LIN {X 0,Y 385.794,Z 704.121,A -85,B 0,C 180,E1 11186.142,E2 11186.142} C_VEL
LIN {X 0,Y 379.875,Z 692.265,A -85,B 0,C 180,E1 11183.296,E2 11183.296} C_VEL
LIN {X 0,Y 374.459,Z 681.957,A -85,B 0,C 180,E1 11180.23,E2 11180.23} C_VEL
LIN {X 0,Y 370.594,Z 674.701,A -85,B 0,C 180,E1 11177.589,E2 11177.589} C_VEL
LIN {X 0,Y 366.819,Z 667.673,A -85,B 0,C 180,E1 11174.362,E2 11174.362} C_VEL
LIN {X 0,Y 365.103,Z 664.56,A -85,B 0,C 180,E1 11172.495,E2 11172.495} C_VEL
LIN {X 0,Y 363.524,Z 661.381,A -85,B 0,C 180,E1 11170.299,E2 11170.299} C_VEL
LIN {X 0,Y 361.927,Z 657.573,A -85,B 0,C 180,E1 11166.663,E2 11166.663} C_VEL
LIN {X 0,Y 361.691,Z 655.978,A -85,B 0,C 180,E1 11161.584,E2 11161.584} C_VEL
LIN {X 0,Y 363.057,Z 656.603,A -85,B 0,C 180,E1 11157.948,E2 11157.948} C_VEL
LIN {X 0,Y 366.472,Z 659.778,A -85,B 0,C 180,E1 11153.498,E2 11153.498} C_VEL
LIN {X 0,Y 370.493,Z 664.801,A -85,B 0,C 180,E1 11149.975,E2 11149.975} C_VEL
LIN {X 0,Y 374.313,Z 669.836,A -85,B 0,C 180,E1 11147.347,E2 11147.347} C_VEL
LIN {X 0,Y 379.523,Z 676.993,A -85,B 0,C 180,E1 11144.372,E2 11144.372} C_VEL
LIN {X 0,Y 385.577,Z 686.162,A -85,B 0,C 180,E1 11141.439,E2 11141.439} C_VEL
LIN {X 0,Y 391.936,Z 696.414,A -85,B 0,C 180,E1 11138.761,E2 11138.761} C_VEL
LIN {X 0,Y 396.859,Z 705.085,A -85,B 0,C 180,E1 11136.889,E2 11136.889} C_VEL
LIN {X 0,Y 378.142,Z 929.621,A -85,B 0,C 180,E1 11132.962,E2 11132.962} C_VEL
LIN {X 0,Y 374.66,Z 954.802,A -85,B 0,C 180,E1 11132.348,E2 11132.348} C_VEL
LIN {X 0,Y 370.716,Z 975.799,A -85,B 0,C 180,E1 11131.66,E2 11131.66} C_VEL
LIN {X 0,Y 365.231,Z 998.846,A -85,B 0,C 180,E1 11130.683,E2 11130.683} C_VEL
LIN {X 0,Y 359.243,Z 1019.879,A -85,B 0,C 180,E1 11129.564,E2 11129.564} C_VEL
LIN {X 0,Y 351.998,Z 1041.518,A -85,B 0,C 180,E1 11128.137,E2 11128.137} C_VEL
LIN {X 0,Y 344.181,Z 1062.128,A -85,B 0,C 180,E1 11126.485,E2 11126.485} C_VEL
LIN {X 0,Y 335.714,Z 1081.84,A -85,B 0,C 180,E1 11124.544,E2 11124.544} C_VEL
LIN {X 0,Y 327.05,Z 1100.424,A -85,B 0,C 180,E1 11122.355,E2 11122.355} C_VEL
LIN {X 0,Y 318.011,Z 1118.05,A -85,B 0,C 180,E1 11119.819,E2 11119.819} C_VEL
LIN {X 0,Y 308.974,Z 1134.8,A -85,B 0,C 180,E1 11116.934,E2 11116.934} C_VEL
LIN {X 0,Y 300.211,Z 1150.077,A -85,B 0,C 180,E1 11113.718,E2 11113.718} C_VEL
LIN {X 0,Y 291.457,Z 1165.019,A -85,B 0,C 180,E1 11109.905,E2 11109.905} C_VEL
LIN {X 0,Y 284.438,Z 1176.9,A -85,B 0,C 180,E1 11106.196,E2 11106.196} C_VEL
LIN {X 0,Y 277.366,Z 1189.144,A -85,B 0,C 180,E1 11101.514,E2 11101.514} C_VEL
LIN {X 0,Y 272.523,Z 1198.075,A -85,B 0,C 180,E1 11097.297,E2 11097.297} C_VEL
LIN {X 0,Y 268.421,Z 1206.484,A -85,B 0,C 180,E1 11092.33,E2 11092.33} C_VEL
LIN {X 0,Y 266.058,Z 1212.321,A -85,B 0,C 180,E1 11087.948,E2 11087.948} C_VEL
LIN {X 0,Y 264.493,Z 1217.601,A -85,B 0,C 180,E1 11082.665,E2 11082.665} C_VEL
LIN {X 0,Y 264.031,Z 1220.449,A -85,B 0,C 180,E1 11078.493,E2 11078.493} C_VEL
LIN {X 0,Y 263.961,Z 1222.135,A -85,B 0,C 180,E1 11074.562,E2 11074.562} C_VEL
LIN {X 0,Y 264,Z 1222.893,A -85,B 0,C 180,E1 11070,E2 11070} C_VEL
LIN {X 0,Y 263.966,Z 1222.194,A -85,B 0,C 180,E1 11065.655,E2 11065.655} C_VEL
LIN {X 0,Y 264.013,Z 1220.547,A -85,B 0,C 180,E1 11061.726,E2 11061.726} C_VEL
LIN {X 0,Y 264.454,Z 1217.74,A -85,B 0,C 180,E1 11057.555,E2 11057.555} C_VEL
LIN {X 0,Y 265.965,Z 1212.541,A -85,B 0,C 180,E1 11052.271,E2 11052.271} C_VEL
LIN {X 0,Y 268.274,Z 1206.745,A -85,B 0,C 180,E1 11047.888,E2 11047.888} C_VEL
LIN {X 0,Y 272.305,Z 1198.419,A -85,B 0,C 180,E1 11042.915,E2 11042.915} C_VEL
LIN {X 0,Y 277.088,Z 1189.533,A -85,B 0,C 180,E1 11038.694,E2 11038.694} C_VEL
LIN {X 0,Y 283.752,Z 1177.976,A -85,B 0,C 180,E1 11034.202,E2 11034.202} C_VEL
LIN {X 0,Y 290.655,Z 1166.202,A -85,B 0,C 180,E1 11030.476,E2 11030.476} C_VEL
LIN {X 0,Y 299.51,Z 1151.115,A -85,B 0,C 180,E1 11026.553,E2 11026.553} C_VEL
LIN {X 0,Y 307.569,Z 1137.016,A -85,B 0,C 180,E1 11023.536,E2 11023.536} C_VEL
LIN {X 0,Y 317.175,Z 1119.387,A -85,B 0,C 180,E1 11020.421,E2 11020.421} C_VEL
LIN {X 0,Y 325.578,Z 1103.038,A -85,B 0,C 180,E1 11018.027,E2 11018.027} C_VEL
LIN {X 0,Y 334.775,Z 1083.58,A -85,B 0,C 180,E1 11015.672,E2 11015.672} C_VEL
LIN {X 0,Y 342.885,Z 1064.882,A -85,B 0,C 180,E1 11013.792,E2 11013.792} C_VEL
LIN {X 0,Y 350.98,Z 1043.855,A -85,B 0,C 180,E1 11012.059,E2 11012.059} C_VEL
LIN {X 0,Y 358.352,Z 1022.299,A -85,B 0,C 180,E1 11010.598,E2 11010.598} C_VEL
LIN {X 0,Y 364.543,Z 1000.723,A -85,B 0,C 180,E1 11009.429,E2 11009.429} C_VEL
LIN {X 0,Y 370.058,Z 978.122,A -85,B 0,C 180,E1 11008.442,E2 11008.442} C_VEL
LIN {X 0,Y 374.312,Z 955.693,A -85,B 0,C 180,E1 11007.695,E2 11007.695} C_VEL
LIN {X 0,Y 377.785,Z 931.228,A -85,B 0,C 180,E1 11007.087,E2 11007.087} C_VEL
LIN {X 0,Y 387.415,Z 815.943,A -85,B 0,C 180,E1 11005.031,E2 11005.031} C_VEL
LIN {X 0,Y 396.675,Z 704.702,A -85,B 0,C 180,E1 11003.116,E2 11003.116} C_VEL
LIN {X 0,Y 389.19,Z 691.96,A -85,B 0,C 180,E1 11000.216,E2 11000.216} C_VEL
LIN {X 0,Y 382.087,Z 680.857,A -85,B 0,C 180,E1 10997.043,E2 10997.043} C_VEL
LIN {X 0,Y 376.158,Z 672.371,A -85,B 0,C 180,E1 10993.92,E2 10993.92} C_VEL
LIN {X 0,Y 372.332,Z 667.309,A -85,B 0,C 180,E1 10991.541,E2 10991.541} C_VEL
LIN {X 0,Y 369.337,Z 663.423,A -85,B 0,C 180,E1 10989.348,E2 10989.348} C_VEL
LIN {X 0,Y 365.813,Z 659.038,A -85,B 0,C 180,E1 10986.119,E2 10986.119} C_VEL
LIN {X 0,Y 362.366,Z 655.946,A -85,B 0,C 180,E1 10981.265,E2 10981.265} C_VEL
LIN {X 0,Y 361.292,Z 655.603,A -85,B 0,C 180,E1 10977.938,E2 10977.938} C_VEL
LIN {X 0,Y 361.77,Z 657.568,A -85,B 0,C 180,E1 10972.696,E2 10972.696} C_VEL
LIN {X 0,Y 363.871,Z 662.416,A -85,B 0,C 180,E1 10968.589,E2 10968.589} C_VEL
LIN {X 0,Y 366.53,Z 667.359,A -85,B 0,C 180,E1 10965.545,E2 10965.545} C_VEL
LIN {X 0,Y 370.214,Z 674.259,A -85,B 0,C 180,E1 10962.392,E2 10962.392} C_VEL
LIN {X 0,Y 373.963,Z 681.257,A -85,B 0,C 180,E1 10959.823,E2 10959.823} C_VEL
LIN {X 0,Y 377.627,Z 688.285,A -85,B 0,C 180,E1 10957.668,E2 10957.668} C_VEL
LIN {X 0,Y 382.471,Z 697.632,A -85,B 0,C 180,E1 10955.191,E2 10955.191} C_VEL
LIN {X 0,Y 388.587,Z 710.276,A -85,B 0,C 180,E1 10952.45,E2 10952.45} C_VEL
LIN {X 0,Y 391.861,Z 717.757,A -85,B 0,C 180,E1 10951.102,E2 10951.102} C_VEL
LIN {X 0,Y 392.576,Z 738.553,A -85,B 0,C 180,E1 10950.077,E2 10950.077} C_VEL
LIN {X 0,Y 377.124,Z 944.509,A -85,B 0,C 180,E1 10946.703,E2 10946.703} C_VEL
LIN {X 0,Y 373.9,Z 967.663,A -85,B 0,C 180,E1 10946.174,E2 10946.174} C_VEL
LIN {X 0,Y 369.642,Z 989.416,A -85,B 0,C 180,E1 10945.52,E2 10945.52} C_VEL
LIN {X 0,Y 364.143,Z 1011.031,A -85,B 0,C 180,E1 10944.636,E2 10944.636} C_VEL
LIN {X 0,Y 357.235,Z 1033.546,A -85,B 0,C 180,E1 10943.444,E2 10943.444} C_VEL
LIN {X 0,Y 350.094,Z 1053.415,A -85,B 0,C 180,E1 10942.117,E2 10942.117} C_VEL
LIN {X 0,Y 342.071,Z 1072.713,A -85,B 0,C 180,E1 10940.503,E2 10940.503} C_VEL
LIN {X 0,Y 333.358,Z 1091.539,A -85,B 0,C 180,E1 10938.576,E2 10938.576} C_VEL
LIN {X 0,Y 324.769,Z 1108.217,A -85,B 0,C 180,E1 10936.471,E2 10936.471} C_VEL
LIN {X 0,Y 315.047,Z 1125.58,A -85,B 0,C 180,E1 10933.778,E2 10933.778} C_VEL
LIN {X 0,Y 306.311,Z 1140.176,A -85,B 0,C 180,E1 10931.003,E2 10931.003} C_VEL
LIN {X 0,Y 297.865,Z 1153.372,A -85,B 0,C 180,E1 10927.9,E2 10927.9} C_VEL
LIN {X 0,Y 289.948,Z 1165.474,A -85,B 0,C 180,E1 10924.44,E2 10924.44} C_VEL
LIN {X 0,Y 282.737,Z 1176.152,A -85,B 0,C 180,E1 10920.613,E2 10920.613} C_VEL
LIN {X 0,Y 275.962,Z 1186.354,A -85,B 0,C 180,E1 10916.002,E2 10916.002} C_VEL
LIN {X 0,Y 271.018,Z 1194.256,A -85,B 0,C 180,E1 10911.422,E2 10911.422} C_VEL
LIN {X 0,Y 267.53,Z 1200.274,A -85,B 0,C 180,E1 10906.725,E2 10906.725} C_VEL
LIN {X 0,Y 265.265,Z 1205.087,A -85,B 0,C 180,E1 10901.524,E2 10901.524} C_VEL
LIN {X 0,Y 264.328,Z 1207.797,A -85,B 0,C 180,E1 10896.952,E2 10896.952} C_VEL
LIN {X 0,Y 264.041,Z 1209.184,A -85,B 0,C 180,E1 10892.17,E2 10892.17} C_VEL
LIN {X 0,Y 264.03,Z 1209.24,A -85,B 0,C 180,E1 10888.264,E2 10888.264} C_VEL
LIN {X 0,Y 264.252,Z 1208.179,A -85,B 0,C 180,E1 10883.7,E2 10883.7} C_VEL
LIN {X 0,Y 265.114,Z 1205.486,A -85,B 0,C 180,E1 10878.911,E2 10878.911} C_VEL
LIN {X 0,Y 267.122,Z 1201.154,A -85,B 0,C 180,E1 10873.92,E2 10873.92} C_VEL
LIN {X 0,Y 270.39,Z 1195.311,A -85,B 0,C 180,E1 10869.207,E2 10869.207} C_VEL
LIN {X 0,Y 275.363,Z 1187.374,A -85,B 0,C 180,E1 10864.399,E2 10864.399} C_VEL
LIN {X 0,Y 281.45,Z 1178.27,A -85,B 0,C 180,E1 10860.094,E2 10860.094} C_VEL
LIN {X 0,Y 288.655,Z 1167.471,A -85,B 0,C 180,E1 10856.105,E2 10856.105} C_VEL
LIN {X 0,Y 297.278,Z 1154.456,A -85,B 0,C 180,E1 10852.256,E2 10852.256} C_VEL
LIN {X 0,Y 306.152,Z 1140.649,A -85,B 0,C 180,E1 10848.971,E2 10848.971} C_VEL
LIN {X 0,Y 314.878,Z 1126.108,A -85,B 0,C 180,E1 10846.193,E2 10846.193} C_VEL
LIN {X 0,Y 324.307,Z 1109.391,A -85,B 0,C 180,E1 10843.571,E2 10843.571} C_VEL
LIN {X 0,Y 332.882,Z 1092.803,A -85,B 0,C 180,E1 10841.456,E2 10841.456} C_VEL
LIN {X 0,Y 341.882,Z 1073.546,A -85,B 0,C 180,E1 10839.459,E2 10839.459} C_VEL
LIN {X 0,Y 349.998,Z 1054.168,A -85,B 0,C 180,E1 10837.825,E2 10837.825} C_VEL
LIN {X 0,Y 357.378,Z 1033.67,A -85,B 0,C 180,E1 10836.452,E2 10836.452} C_VEL
LIN {X 0,Y 364.292,Z 1011.192,A -85,B 0,C 180,E1 10835.261,E2 10835.261} C_VEL
LIN {X 0,Y 369.611,Z 990.338,A -85,B 0,C 180,E1 10834.404,E2 10834.404} C_VEL
LIN {X 0,Y 374.035,Z 968.047,A -85,B 0,C 180,E1 10833.728,E2 10833.728} C_VEL
LIN {X 0,Y 377.274,Z 945.089,A -85,B 0,C 180,E1 10833.2,E2 10833.2} C_VEL
LIN {X 0,Y 385.345,Z 837.315,A -85,B 0,C 180,E1 10831.408,E2 10831.408} C_VEL
LIN {X 0,Y 392.815,Z 736.753,A -85,B 0,C 180,E1 10829.76,E2 10829.76} C_VEL
LIN {X 0,Y 392.625,Z 732.027,A -85,B 0,C 180,E1 10829.521,E2 10829.521} C_VEL
LIN {X 0,Y 392.068,Z 728.255,A -85,B 0,C 180,E1 10829.205,E2 10829.205} C_VEL
LIN {X 0,Y 390.556,Z 724.358,A -85,B 0,C 180,E1 10828.585,E2 10828.585} C_VEL
LIN {X 0,Y 386.327,Z 717.157,A -85,B 0,C 180,E1 10826.909,E2 10826.909} C_VEL
LIN {X 0,Y 380.447,Z 704.585,A -85,B 0,C 180,E1 10824.164,E2 10824.164} C_VEL
LIN {X 0,Y 375.315,Z 694.392,A -85,B 0,C 180,E1 10821.407,E2 10821.407} C_VEL
LIN {X 0,Y 371.624,Z 687.152,A -85,B 0,C 180,E1 10819.081,E2 10819.081} C_VEL
LIN {X 0,Y 368.331,Z 680.76,A -85,B 0,C 180,E1 10816.634,E2 10816.634} C_VEL
LIN {X 0,Y 364.751,Z 673.725,A -85,B 0,C 180,E1 10813.232,E2 10813.232} C_VEL
LIN {X 0,Y 362.352,Z 669.116,A -85,B 0,C 180,E1 10810.012,E2 10810.012} C_VEL
LIN {X 0,Y 360.908,Z 665.464,A -85,B 0,C 180,E1 10806.522,E2 10806.522} C_VEL
LIN {X 0,Y 360.716,Z 663.92,A -85,B 0,C 180,E1 10801.588,E2 10801.588} C_VEL
LIN {X 0,Y 362.079,Z 664.569,A -85,B 0,C 180,E1 10797.943,E2 10797.943} C_VEL
LIN {X 0,Y 365.256,Z 667.574,A -85,B 0,C 180,E1 10793.713,E2 10793.713} C_VEL
LIN {X 0,Y 369.182,Z 672.629,A -85,B 0,C 180,E1 10790.176,E2 10790.176} C_VEL
LIN {X 0,Y 372.704,Z 677.357,A -85,B 0,C 180,E1 10787.685,E2 10787.685} C_VEL
LIN {X 0,Y 377.735,Z 684.444,A -85,B 0,C 180,E1 10784.729,E2 10784.729} C_VEL
LIN {X 0,Y 383.502,Z 693.396,A -85,B 0,C 180,E1 10781.846,E2 10781.846} C_VEL
LIN {X 0,Y 389.565,Z 703.408,A -85,B 0,C 180,E1 10779.216,E2 10779.216} C_VEL
LIN {X 0,Y 392.961,Z 709.665,A -85,B 0,C 180,E1 10777.857,E2 10777.857} C_VEL
LIN {X 0,Y 374.215,Z 929.569,A -85,B 0,C 180,E1 10774.027,E2 10774.027} C_VEL
LIN {X 0,Y 370.645,Z 954.977,A -85,B 0,C 180,E1 10773.413,E2 10773.413} C_VEL
LIN {X 0,Y 366.64,Z 975.871,A -85,B 0,C 180,E1 10772.734,E2 10772.734} C_VEL
LIN {X 0,Y 360.947,Z 999.256,A -85,B 0,C 180,E1 10771.75,E2 10771.75} C_VEL
LIN {X 0,Y 355.065,Z 1019.451,A -85,B 0,C 180,E1 10770.685,E2 10770.685} C_VEL
LIN {X 0,Y 347.402,Z 1041.849,A -85,B 0,C 180,E1 10769.217,E2 10769.217} C_VEL
LIN {X 0,Y 339.431,Z 1062.322,A -85,B 0,C 180,E1 10767.579,E2 10767.579} C_VEL
LIN {X 0,Y 330.689,Z 1082.093,A -85,B 0,C 180,E1 10765.632,E2 10765.632} C_VEL
LIN {X 0,Y 321.475,Z 1101.221,A -85,B 0,C 180,E1 10763.363,E2 10763.363} C_VEL
LIN {X 0,Y 312.175,Z 1118.751,A -85,B 0,C 180,E1 10760.813,E2 10760.813} C_VEL
LIN {X 0,Y 302.457,Z 1136.035,A -85,B 0,C 180,E1 10757.774,E2 10757.774} C_VEL
LIN {X 0,Y 293.558,Z 1150.996,A -85,B 0,C 180,E1 10754.558,E2 10754.558} C_VEL
LIN {X 0,Y 284.306,Z 1166.072,A -85,B 0,C 180,E1 10750.588,E2 10750.588} C_VEL
LIN {X 0,Y 276.716,Z 1178.428,A -85,B 0,C 180,E1 10746.598,E2 10746.598} C_VEL
LIN {X 0,Y 270.039,Z 1189.39,A -85,B 0,C 180,E1 10742.221,E2 10742.221} C_VEL
LIN {X 0,Y 264.749,Z 1198.691,A -85,B 0,C 180,E1 10737.679,E2 10737.679} C_VEL
LIN {X 0,Y 260.66,Z 1206.584,A -85,B 0,C 180,E1 10732.794,E2 10732.794} C_VEL
LIN {X 0,Y 258.073,Z 1212.639,A -85,B 0,C 180,E1 10728.056,E2 10728.056} C_VEL
LIN {X 0,Y 256.518,Z 1217.562,A -85,B 0,C 180,E1 10722.837,E2 10722.837} C_VEL
LIN {X 0,Y 256.034,Z 1220.362,A -85,B 0,C 180,E1 10718.534,E2 10718.534} C_VEL
LIN {X 0,Y 255.964,Z 1222.002,A -85,B 0,C 180,E1 10714.481,E2 10714.481} C_VEL
LIN {X 0,Y 256.002,Z 1222.689,A -85,B 0,C 180,E1 10710,E2 10710} C_VEL
LIN {X 0,Y 255.964,Z 1221.989,A -85,B 0,C 180,E1 10705.519,E2 10705.519} C_VEL
LIN {X 0,Y 256.034,Z 1220.34,A -85,B 0,C 180,E1 10701.466,E2 10701.466} C_VEL
LIN {X 0,Y 256.547,Z 1217.411,A -85,B 0,C 180,E1 10697.002,E2 10697.002} C_VEL
LIN {X 0,Y 258.235,Z 1212.14,A -85,B 0,C 180,E1 10691.559,E2 10691.559} C_VEL
LIN {X 0,Y 260.857,Z 1206.118,A -85,B 0,C 180,E1 10686.919,E2 10686.919} C_VEL
LIN {X 0,Y 265.42,Z 1197.347,A -85,B 0,C 180,E1 10681.663,E2 10681.663} C_VEL
LIN {X 0,Y 270.607,Z 1188.348,A -85,B 0,C 180,E1 10677.354,E2 10677.354} C_VEL
LIN {X 0,Y 277.762,Z 1176.54,A -85,B 0,C 180,E1 10672.789,E2 10672.789} C_VEL
LIN {X 0,Y 285.492,Z 1164.055,A -85,B 0,C 180,E1 10668.852,E2 10668.852} C_VEL
LIN {X 0,Y 294.012,Z 1150.038,A -85,B 0,C 180,E1 10665.255,E2 10665.255} C_VEL
LIN {X 0,Y 302.957,Z 1134.986,A -85,B 0,C 180,E1 10662.049,E2 10662.049} C_VEL
LIN {X 0,Y 312.152,Z 1118.527,A -85,B 0,C 180,E1 10659.181,E2 10659.181} C_VEL
LIN {X 0,Y 321.452,Z 1100.971,A -85,B 0,C 180,E1 10656.631,E2 10656.631} C_VEL
LIN {X 0,Y 330.664,Z 1081.784,A -85,B 0,C 180,E1 10654.362,E2 10654.362} C_VEL
LIN {X 0,Y 339.301,Z 1062.196,A -85,B 0,C 180,E1 10652.435,E2 10652.435} C_VEL
LIN {X 0,Y 347.374,Z 1041.433,A -85,B 0,C 180,E1 10650.775,E2 10650.775} C_VEL
LIN {X 0,Y 355.283,Z 1018.102,A -85,B 0,C 180,E1 10649.259,E2 10649.259} C_VEL
LIN {X 0,Y 361.423,Z 996.801,A -85,B 0,C 180,E1 10648.151,E2 10648.151} C_VEL
LIN {X 0,Y 366.99,Z 973.192,A -85,B 0,C 180,E1 10647.189,E2 10647.189} C_VEL
LIN {X 0,Y 370.984,Z 951.918,A -85,B 0,C 180,E1 10646.519,E2 10646.519} C_VEL
LIN {X 0,Y 374.217,Z 927.542,A -85,B 0,C 180,E1 10645.952,E2 10645.952} C_VEL
LIN {X 0,Y 392.786,Z 709.176,A -85,B 0,C 180,E1 10642.143,E2 10642.143} C_VEL
LIN {X 0,Y 386.129,Z 697.783,A -85,B 0,C 180,E1 10639.436,E2 10639.436} C_VEL
LIN {X 0,Y 380.016,Z 687.987,A -85,B 0,C 180,E1 10636.588,E2 10636.588} C_VEL
LIN {X 0,Y 374.376,Z 679.738,A -85,B 0,C 180,E1 10633.515,E2 10633.515} C_VEL
LIN {X 0,Y 370.879,Z 674.979,A -85,B 0,C 180,E1 10631.272,E2 10631.272} C_VEL
LIN {X 0,Y 367.952,Z 671.114,A -85,B 0,C 180,E1 10629.068,E2 10629.068} C_VEL
LIN {X 0,Y 364.525,Z 666.807,A -85,B 0,C 180,E1 10625.825,E2 10625.825} C_VEL
LIN {X 0,Y 361.316,Z 663.84,A -85,B 0,C 180,E1 10621.11,E2 10621.11} C_VEL
LIN {X 0,Y 360.292,Z 663.572,A -85,B 0,C 180,E1 10617.773,E2 10617.773} C_VEL
LIN {X 0,Y 360.787,Z 665.64,A -85,B 0,C 180,E1 10612.676,E2 10612.676} C_VEL
LIN {X 0,Y 362.729,Z 670.25,A -85,B 0,C 180,E1 10608.794,E2 10608.794} C_VEL
LIN {X 0,Y 365.321,Z 675.211,A -85,B 0,C 180,E1 10605.739,E2 10605.739} C_VEL
LIN {X 0,Y 369.966,Z 684.06,A -85,B 0,C 180,E1 10601.811,E2 10601.811} C_VEL
LIN {X 0,Y 374.756,Z 693.471,A -85,B 0,C 180,E1 10598.683,E2 10598.683} C_VEL
LIN {X 0,Y 379.179,Z 702.42,A -85,B 0,C 180,E1 10596.247,E2 10596.247} C_VEL
LIN {X 0,Y 384.53,Z 713.605,A -85,B 0,C 180,E1 10593.682,E2 10593.682} C_VEL
LIN {X 0,Y 388.454,Z 722.612,A -85,B 0,C 180,E1 10591.972,E2 10591.972} C_VEL
LIN {X 0,Y 388.937,Z 740.008,A -85,B 0,C 180,E1 10591.109,E2 10591.109} C_VEL
LIN {X 0,Y 373.161,Z 944.254,A -85,B 0,C 180,E1 10587.769,E2 10587.769} C_VEL
LIN {X 0,Y 369.873,Z 967.387,A -85,B 0,C 180,E1 10587.244,E2 10587.244} C_VEL
LIN {X 0,Y 365.386,Z 989.729,A -85,B 0,C 180,E1 10586.576,E2 10586.576} C_VEL
LIN {X 0,Y 359.955,Z 1010.634,A -85,B 0,C 180,E1 10585.728,E2 10585.728} C_VEL
LIN {X 0,Y 352.896,Z 1033.203,A -85,B 0,C 180,E1 10584.545,E2 10584.545} C_VEL
LIN {X 0,Y 345.682,Z 1052.843,A -85,B 0,C 180,E1 10583.245,E2 10583.245} C_VEL
LIN {X 0,Y 337.362,Z 1072.447,A -85,B 0,C 180,E1 10581.62,E2 10581.62} C_VEL
LIN {X 0,Y 328.535,Z 1091.091,A -85,B 0,C 180,E1 10579.724,E2 10579.724} C_VEL
LIN {X 0,Y 319.576,Z 1108.021,A -85,B 0,C 180,E1 10577.593,E2 10577.593} C_VEL
LIN {X 0,Y 309.826,Z 1124.972,A -85,B 0,C 180,E1 10574.971,E2 10574.971} C_VEL
LIN {X 0,Y 300.767,Z 1139.633,A -85,B 0,C 180,E1 10572.184,E2 10572.184} C_VEL
LIN {X 0,Y 291.981,Z 1152.942,A -85,B 0,C 180,E1 10569.057,E2 10569.057} C_VEL
LIN {X 0,Y 283.703,Z 1165.143,A -85,B 0,C 180,E1 10565.557,E2 10565.557} C_VEL
LIN {X 0,Y 275.782,Z 1176.382,A -85,B 0,C 180,E1 10561.472,E2 10561.472} C_VEL
LIN {X 0,Y 268.962,Z 1186.184,A -85,B 0,C 180,E1 10556.97,E2 10556.97} C_VEL
LIN {X 0,Y 263.689,Z 1194.143,A -85,B 0,C 180,E1 10552.283,E2 10552.283} C_VEL
LIN {X 0,Y 259.898,Z 1200.284,A -85,B 0,C 180,E1 10547.423,E2 10547.423} C_VEL
LIN {X 0,Y 257.508,Z 1204.99,A -85,B 0,C 180,E1 10542.331,E2 10542.331} C_VEL
LIN {X 0,Y 256.415,Z 1207.787,A -85,B 0,C 180,E1 10537.619,E2 10537.619} C_VEL
LIN {X 0,Y 256.056,Z 1209.346,A -85,B 0,C 180,E1 10532.686,E2 10532.686} C_VEL
LIN {X 0,Y 256.03,Z 1209.466,A -85,B 0,C 180,E1 10528.434,E2 10528.434} C_VEL
LIN {X 0,Y 256.23,Z 1208.515,A -85,B 0,C 180,E1 10523.952,E2 10523.952} C_VEL
LIN {X 0,Y 257.079,Z 1205.997,A -85,B 0,C 180,E1 10519.014,E2 10519.014} C_VEL
LIN {X 0,Y 259.065,Z 1201.929,A -85,B 0,C 180,E1 10513.955,E2 10513.955} C_VEL
LIN {X 0,Y 262.508,Z 1196.005,A -85,B 0,C 180,E1 10508.941,E2 10508.941} C_VEL
LIN {X 0,Y 267.799,Z 1187.982,A -85,B 0,C 180,E1 10503.86,E2 10503.86} C_VEL
LIN {X 0,Y 273.997,Z 1179.111,A -85,B 0,C 180,E1 10499.52,E2 10499.52} C_VEL
LIN {X 0,Y 281.17,Z 1168.821,A -85,B 0,C 180,E1 10495.569,E2 10495.569} C_VEL
LIN {X 0,Y 289.565,Z 1156.76,A -85,B 0,C 180,E1 10491.824,E2 10491.824} C_VEL
LIN {X 0,Y 298.078,Z 1143.937,A -85,B 0,C 180,E1 10488.639,E2 10488.639} C_VEL
LIN {X 0,Y 308.009,Z 1128.22,A -85,B 0,C 180,E1 10485.479,E2 10485.479} C_VEL
LIN {X 0,Y 317.057,Z 1112.892,A -85,B 0,C 180,E1 10482.977,E2 10482.977} C_VEL
LIN {X 0,Y 326.366,Z 1095.595,A -85,B 0,C 180,E1 10480.691,E2 10480.691} C_VEL
LIN {X 0,Y 335.235,Z 1077.624,A -85,B 0,C 180,E1 10478.745,E2 10478.745} C_VEL
LIN {X 0,Y 343.461,Z 1058.717,A -85,B 0,C 180,E1 10477.094,E2 10477.094} C_VEL
LIN {X 0,Y 351.653,Z 1037.304,A -85,B 0,C 180,E1 10475.592,E2 10475.592} C_VEL
LIN {X 0,Y 358.331,Z 1017.005,A -85,B 0,C 180,E1 10474.458,E2 10474.458} C_VEL
LIN {X 0,Y 364.077,Z 995.81,A -85,B 0,C 180,E1 10473.541,E2 10473.541} C_VEL
LIN {X 0,Y 368.978,Z 973.69,A -85,B 0,C 180,E1 10472.811,E2 10472.811} C_VEL
LIN {X 0,Y 372.498,Z 951.44,A -85,B 0,C 180,E1 10472.272,E2 10472.272} C_VEL
LIN {X 0,Y 375.283,Z 921.525,A -85,B 0,C 180,E1 10471.727,E2 10471.727} C_VEL
LIN {X 0,Y 389.201,Z 738.35,A -85,B 0,C 180,E1 10468.732,E2 10468.732} C_VEL
LIN {X 0,Y 388.611,Z 722.277,A -85,B 0,C 180,E1 10467.881,E2 10467.881} C_VEL
LIN {X 0,Y 386.327,Z 717.157,A -85,B 0,C 180,E1 10466.909,E2 10466.909} C_VEL
LIN {X 0,Y 384.392,Z 713.944,A -85,B 0,C 180,E1 10466.094,E2 10466.094} C_VEL
LIN {X 0,Y 380.9,Z 710.969,A -85,B 0,C 180,E1 10464.659,E2 10464.659} C_VEL
LIN {X 0,Y 376.857,Z 707.794,A -85,B 0,C 180,E1 10462.854,E2 10462.854} C_VEL
LIN {X 0,Y 375.422,Z 705.527,A -85,B 0,C 180,E1 10462.102,E2 10462.102} C_VEL
LIN {X 0,Y 370.638,Z 695.84,A -85,B 0,C 180,E1 10459.134,E2 10459.134} C_VEL
LIN {X 0,Y 367.17,Z 688.895,A -85,B 0,C 180,E1 10456.534,E2 10456.534} C_VEL
LIN {X 0,Y 363.695,Z 681.889,A -85,B 0,C 180,E1 10453.191,E2 10453.191} C_VEL
LIN {X 0,Y 361.254,Z 676.958,A -85,B 0,C 180,E1 10449.832,E2 10449.832} C_VEL
LIN {X 0,Y 359.891,Z 673.355,A -85,B 0,C 180,E1 10446.381,E2 10446.381} C_VEL
LIN {X 0,Y 359.776,Z 671.849,A -85,B 0,C 180,E1 10441.433,E2 10441.433} C_VEL
LIN {X 0,Y 361.101,Z 672.54,A -85,B 0,C 180,E1 10437.937,E2 10437.937} C_VEL
LIN {X 0,Y 364.103,Z 675.49,A -85,B 0,C 180,E1 10433.852,E2 10433.852} C_VEL
LIN {X 0,Y 367.782,Z 680.304,A -85,B 0,C 180,E1 10430.454,E2 10430.454} C_VEL
LIN {X 0,Y 371.219,Z 685.052,A -85,B 0,C 180,E1 10427.951,E2 10427.951} C_VEL
LIN {X 0,Y 375.96,Z 691.894,A -85,B 0,C 180,E1 10425.089,E2 10425.089} C_VEL
LIN {X 0,Y 381.447,Z 700.629,A -85,B 0,C 180,E1 10422.258,E2 10422.258} C_VEL
LIN {X 0,Y 387.22,Z 710.4,A -85,B 0,C 180,E1 10419.677,E2 10419.677} C_VEL
LIN {X 0,Y 389.192,Z 714.231,A -85,B 0,C 180,E1 10418.845,E2 10418.845} C_VEL
LIN {X 0,Y 370.318,Z 930.496,A -85,B 0,C 180,E1 10415.094,E2 10415.094} C_VEL
LIN {X 0,Y 366.698,Z 955.504,A -85,B 0,C 180,E1 10414.491,E2 10414.491} C_VEL
LIN {X 0,Y 362.562,Z 976.573,A -85,B 0,C 180,E1 10413.81,E2 10413.81} C_VEL
LIN {X 0,Y 356.791,Z 999.672,A -85,B 0,C 180,E1 10412.841,E2 10412.841} C_VEL
LIN {X 0,Y 350.52,Z 1020.669,A -85,B 0,C 180,E1 10411.736,E2 10411.736} C_VEL
LIN {X 0,Y 342.933,Z 1042.18,A -85,B 0,C 180,E1 10410.325,E2 10410.325} C_VEL
LIN {X 0,Y 334.693,Z 1062.801,A -85,B 0,C 180,E1 10408.68,E2 10408.68} C_VEL
LIN {X 0,Y 325.79,Z 1082.351,A -85,B 0,C 180,E1 10406.752,E2 10406.752} C_VEL
LIN {X 0,Y 316.311,Z 1101.432,A -85,B 0,C 180,E1 10404.484,E2 10404.484} C_VEL
LIN {X 0,Y 306.754,Z 1118.882,A -85,B 0,C 180,E1 10401.936,E2 10401.936} C_VEL
LIN {X 0,Y 296.949,Z 1135.743,A -85,B 0,C 180,E1 10398.958,E2 10398.958} C_VEL
LIN {X 0,Y 288.192,Z 1149.926,A -85,B 0,C 180,E1 10395.903,E2 10395.903} C_VEL
LIN {X 0,Y 278.908,Z 1164.528,A -85,B 0,C 180,E1 10392.089,E2 10392.089} C_VEL
LIN {X 0,Y 271.126,Z 1176.523,A -85,B 0,C 180,E1 10388.23,E2 10388.23} C_VEL
LIN {X 0,Y 263.235,Z 1188.871,A -85,B 0,C 180,E1 10383.315,E2 10383.315} C_VEL
LIN {X 0,Y 257.623,Z 1198.157,A -85,B 0,C 180,E1 10378.699,E2 10378.699} C_VEL
LIN {X 0,Y 253.08,Z 1206.368,A -85,B 0,C 180,E1 10373.517,E2 10373.517} C_VEL
LIN {X 0,Y 250.289,Z 1212.426,A -85,B 0,C 180,E1 10368.638,E2 10368.638} C_VEL
LIN {X 0,Y 248.59,Z 1217.356,A -85,B 0,C 180,E1 10363.248,E2 10363.248} C_VEL
LIN {X 0,Y 248.056,Z 1220.155,A -85,B 0,C 180,E1 10358.811,E2 10358.811} C_VEL
LIN {X 0,Y 247.967,Z 1221.869,A -85,B 0,C 180,E1 10354.394,E2 10354.394} C_VEL
LIN {X 0,Y 247.996,Z 1222.465,A -85,B 0,C 180,E1 10349.769,E2 10349.769} C_VEL
LIN {X 0,Y 247.962,Z 1221.783,A -85,B 0,C 180,E1 10345.374,E2 10345.374} C_VEL
LIN {X 0,Y 248.056,Z 1220.133,A -85,B 0,C 180,E1 10341.189,E2 10341.189} C_VEL
LIN {X 0,Y 248.639,Z 1217.152,A -85,B 0,C 180,E1 10336.512,E2 10336.512} C_VEL
LIN {X 0,Y 250.498,Z 1211.842,A -85,B 0,C 180,E1 10330.895,E2 10330.895} C_VEL
LIN {X 0,Y 253.413,Z 1205.672,A -85,B 0,C 180,E1 10326.022,E2 10326.022} C_VEL
LIN {X 0,Y 258.162,Z 1197.117,A -85,B 0,C 180,E1 10320.791,E2 10320.791} C_VEL
LIN {X 0,Y 263.658,Z 1188.115,A -85,B 0,C 180,E1 10316.381,E2 10316.381} C_VEL
LIN {X 0,Y 271.188,Z 1176.29,A -85,B 0,C 180,E1 10311.727,E2 10311.727} C_VEL
LIN {X 0,Y 279.345,Z 1163.723,A -85,B 0,C 180,E1 10307.708,E2 10307.708} C_VEL
LIN {X 0,Y 288.175,Z 1149.754,A -85,B 0,C 180,E1 10304.093,E2 10304.093} C_VEL
LIN {X 0,Y 297.469,Z 1134.688,A -85,B 0,C 180,E1 10300.863,E2 10300.863} C_VEL
LIN {X 0,Y 307.282,Z 1117.67,A -85,B 0,C 180,E1 10297.902,E2 10297.902} C_VEL
LIN {X 0,Y 316.903,Z 1099.984,A -85,B 0,C 180,E1 10295.354,E2 10295.354} C_VEL
LIN {X 0,Y 326.089,Z 1081.352,A -85,B 0,C 180,E1 10293.168,E2 10293.168} C_VEL
LIN {X 0,Y 335.361,Z 1060.697,A -85,B 0,C 180,E1 10291.166,E2 10291.166} C_VEL
LIN {X 0,Y 342.906,Z 1041.753,A -85,B 0,C 180,E1 10289.667,E2 10289.667} C_VEL
LIN {X 0,Y 350.9,Z 1018.797,A -85,B 0,C 180,E1 10288.178,E2 10288.178} C_VEL
LIN {X 0,Y 357.122,Z 997.753,A -85,B 0,C 180,E1 10287.086,E2 10287.086} C_VEL
LIN {X 0,Y 362.943,Z 973.755,A -85,B 0,C 180,E1 10286.109,E2 10286.109} C_VEL
LIN {X 0,Y 366.967,Z 952.842,A -85,B 0,C 180,E1 10285.453,E2 10285.453} C_VEL
LIN {X 0,Y 370.349,Z 928.156,A -85,B 0,C 180,E1 10284.878,E2 10284.878} C_VEL
LIN {X 0,Y 388.995,Z 713.751,A -85,B 0,C 180,E1 10281.151,E2 10281.151} C_VEL
LIN {X 0,Y 382.618,Z 702.622,A -85,B 0,C 180,E1 10278.394,E2 10278.394} C_VEL
LIN {X 0,Y 376.716,Z 693.273,A -85,B 0,C 180,E1 10275.471,E2 10275.471} C_VEL
LIN {X 0,Y 372.01,Z 686.302,A -85,B 0,C 180,E1 10272.733,E2 10272.733} C_VEL
LIN {X 0,Y 369.218,Z 682.39,A -85,B 0,C 180,E1 10270.849,E2 10270.849} C_VEL
LIN {X 0,Y 366.576,Z 678.803,A -85,B 0,C 180,E1 10268.786,E2 10268.786} C_VEL
LIN {X 0,Y 363.392,Z 674.681,A -85,B 0,C 180,E1 10265.685,E2 10265.685} C_VEL
LIN {X 0,Y 360.334,Z 671.789,A -85,B 0,C 180,E1 10261.113,E2 10261.113} C_VEL
LIN {X 0,Y 359.316,Z 671.52,A -85,B 0,C 180,E1 10257.767,E2 10257.767} C_VEL
LIN {X 0,Y 359.757,Z 673.548,A -85,B 0,C 180,E1 10252.815,E2 10252.815} C_VEL
LIN {X 0,Y 361.641,Z 678.199,A -85,B 0,C 180,E1 10248.929,E2 10248.929} C_VEL
LIN {X 0,Y 364.117,Z 683.066,A -85,B 0,C 180,E1 10245.935,E2 10245.935} C_VEL
LIN {X 0,Y 368.413,Z 691.567,A -85,B 0,C 180,E1 10242.181,E2 10242.181} C_VEL
LIN {X 0,Y 372.883,Z 700.646,A -85,B 0,C 180,E1 10239.147,E2 10239.147} C_VEL
LIN {X 0,Y 377.184,Z 709.607,A -85,B 0,C 180,E1 10236.693,E2 10236.693} C_VEL
LIN {X 0,Y 382.487,Z 721.091,A -85,B 0,C 180,E1 10234.069,E2 10234.069} C_VEL
LIN {X 0,Y 385.14,Z 727.562,A -85,B 0,C 180,E1 10232.853,E2 10232.853} C_VEL
LIN {X 0,Y 385.421,Z 741.52,A -85,B 0,C 180,E1 10232.16,E2 10232.16} C_VEL
LIN {X 0,Y 369.346,Z 943.824,A -85,B 0,C 180,E1 10228.861,E2 10228.861} C_VEL
LIN {X 0,Y 365.988,Z 967.055,A -85,B 0,C 180,E1 10228.339,E2 10228.339} C_VEL
LIN {X 0,Y 361.445,Z 989.3,A -85,B 0,C 180,E1 10227.682,E2 10227.682} C_VEL
LIN {X 0,Y 355.901,Z 1010.235,A -85,B 0,C 180,E1 10226.845,E2 10226.845} C_VEL
LIN {X 0,Y 349.049,Z 1031.86,A -85,B 0,C 180,E1 10225.732,E2 10225.732} C_VEL
LIN {X 0,Y 342.003,Z 1050.74,A -85,B 0,C 180,E1 10224.509,E2 10224.509} C_VEL
LIN {X 0,Y 333.459,Z 1070.723,A -85,B 0,C 180,E1 10222.9,E2 10222.9} C_VEL
LIN {X 0,Y 324.594,Z 1089.188,A -85,B 0,C 180,E1 10221.067,E2 10221.067} C_VEL
LIN {X 0,Y 315.124,Z 1106.73,A -85,B 0,C 180,E1 10218.9,E2 10218.9} C_VEL
LIN {X 0,Y 305.321,Z 1123.458,A -85,B 0,C 180,E1 10216.363,E2 10216.363} C_VEL
LIN {X 0,Y 296.42,Z 1137.433,A -85,B 0,C 180,E1 10213.748,E2 10213.748} C_VEL
LIN {X 0,Y 286.225,Z 1152.513,A -85,B 0,C 180,E1 10210.259,E2 10210.259} C_VEL
LIN {X 0,Y 277.571,Z 1164.779,A -85,B 0,C 180,E1 10206.724,E2 10206.724} C_VEL
LIN {X 0,Y 269.621,Z 1175.61,A -85,B 0,C 180,E1 10202.78,E2 10202.78} C_VEL
LIN {X 0,Y 262.637,Z 1185.227,A -85,B 0,C 180,E1 10198.416,E2 10198.416} C_VEL
LIN {X 0,Y 257.087,Z 1192.996,A -85,B 0,C 180,E1 10193.858,E2 10193.858} C_VEL
LIN {X 0,Y 252.508,Z 1199.966,A -85,B 0,C 180,E1 10188.468,E2 10188.468} C_VEL
LIN {X 0,Y 249.883,Z 1204.71,A -85,B 0,C 180,E1 10183.419,E2 10183.419} C_VEL
LIN {X 0,Y 248.523,Z 1207.778,A -85,B 0,C 180,E1 10178.328,E2 10178.328} C_VEL
LIN {X 0,Y 248.081,Z 1209.452,A -85,B 0,C 180,E1 10173.466,E2 10173.466} C_VEL
LIN {X 0,Y 248.03,Z 1209.708,A -85,B 0,C 180,E1 10168.79,E2 10168.79} C_VEL
LIN {X 0,Y 248.19,Z 1208.911,A -85,B 0,C 180,E1 10164.452,E2 10164.452} C_VEL
LIN {X 0,Y 249.05,Z 1206.507,A -85,B 0,C 180,E1 10159.124,E2 10159.124} C_VEL
LIN {X 0,Y 250.858,Z 1202.851,A -85,B 0,C 180,E1 10154.274,E2 10154.274} C_VEL
LIN {X 0,Y 254.315,Z 1197.191,A -85,B 0,C 180,E1 10149.037,E2 10149.037} C_VEL
LIN {X 0,Y 259.208,Z 1190.129,A -85,B 0,C 180,E1 10144.159,E2 10144.159} C_VEL
LIN {X 0,Y 265.45,Z 1181.422,A -85,B 0,C 180,E1 10139.609,E2 10139.609} C_VEL
LIN {X 0,Y 273.312,Z 1170.73,A -85,B 0,C 180,E1 10135.201,E2 10135.201} C_VEL
LIN {X 0,Y 281.404,Z 1159.554,A -85,B 0,C 180,E1 10131.553,E2 10131.553} C_VEL
LIN {X 0,Y 291.031,Z 1145.708,A -85,B 0,C 180,E1 10127.938,E2 10127.938} C_VEL
LIN {X 0,Y 300.635,Z 1131.24,A -85,B 0,C 180,E1 10124.895,E2 10124.895} C_VEL
LIN {X 0,Y 310.125,Z 1115.698,A -85,B 0,C 180,E1 10122.276,E2 10122.276} C_VEL
LIN {X 0,Y 320.241,Z 1097.763,A -85,B 0,C 180,E1 10119.82,E2 10119.82} C_VEL
LIN {X 0,Y 328.955,Z 1080.743,A -85,B 0,C 180,E1 10117.931,E2 10117.931} C_VEL
LIN {X 0,Y 337.672,Z 1061.624,A -85,B 0,C 180,E1 10116.208,E2 10116.208} C_VEL
LIN {X 0,Y 345.669,Z 1041.904,A -85,B 0,C 180,E1 10114.767,E2 10114.767} C_VEL
LIN {X 0,Y 352.795,Z 1021.117,A -85,B 0,C 180,E1 10113.569,E2 10113.569} C_VEL
LIN {X 0,Y 359.15,Z 999.248,A -85,B 0,C 180,E1 10112.578,E2 10112.578} C_VEL
LIN {X 0,Y 364.056,Z 978.295,A -85,B 0,C 180,E1 10111.861,E2 10111.861} C_VEL
LIN {X 0,Y 368.158,Z 954.793,A -85,B 0,C 180,E1 10111.262,E2 10111.262} C_VEL
LIN {X 0,Y 370.725,Z 931.676,A -85,B 0,C 180,E1 10110.81,E2 10110.81} C_VEL
LIN {X 0,Y 385.711,Z 739.836,A -85,B 0,C 180,E1 10107.68,E2 10107.68} C_VEL
LIN {X 0,Y 385.319,Z 727.254,A -85,B 0,C 180,E1 10107.008,E2 10107.008} C_VEL
LIN {X 0,Y 380.001,Z 715.293,A -85,B 0,C 180,E1 10104.525,E2 10104.525} C_VEL
LIN {X 0,Y 375.422,Z 705.527,A -85,B 0,C 180,E1 10102.102,E2 10102.102} C_VEL
LIN {X 0,Y 373.482,Z 702.765,A -85,B 0,C 180,E1 10101.036,E2 10101.036} C_VEL
LIN {X 0,Y 370.031,Z 700.894,A -85,B 0,C 180,E1 10099.147,E2 10099.147} C_VEL
LIN {X 0,Y 367.214,Z 699.116,A -85,B 0,C 180,E1 10097.381,E2 10097.381} C_VEL
LIN {X 0,Y 366.559,Z 698.136,A -85,B 0,C 180,E1 10096.887,E2 10096.887} C_VEL
LIN {X 0,Y 362.784,Z 690.359,A -85,B 0,C 180,E1 10093.305,E2 10093.305} C_VEL
LIN {X 0,Y 360.324,Z 685.05,A -85,B 0,C 180,E1 10089.907,E2 10089.907} C_VEL
LIN {X 0,Y 358.848,Z 681.171,A -85,B 0,C 180,E1 10086.078,E2 10086.078} C_VEL
LIN {X 0,Y 358.837,Z 679.779,A -85,B 0,C 180,E1 10081.277,E2 10081.277} C_VEL
LIN {X 0,Y 360.123,Z 680.513,A -85,B 0,C 180,E1 10077.931,E2 10077.931} C_VEL
LIN {X 0,Y 362.865,Z 683.226,A -85,B 0,C 180,E1 10074.107,E2 10074.107} C_VEL
LIN {X 0,Y 366.483,Z 688.128,A -85,B 0,C 180,E1 10070.657,E2 10070.657} C_VEL
LIN {X 0,Y 369.747,Z 692.744,A -85,B 0,C 180,E1 10068.219,E2 10068.219} C_VEL
LIN {X 0,Y 374.197,Z 699.341,A -85,B 0,C 180,E1 10065.453,E2 10065.453} C_VEL
LIN {X 0,Y 379.561,Z 708.109,A -85,B 0,C 180,E1 10062.603,E2 10062.603} C_VEL
LIN {X 0,Y 385.062,Z 717.69,A -85,B 0,C 180,E1 10060.073,E2 10060.073} C_VEL
LIN {X 0,Y 385.54,Z 718.856,A -85,B 0,C 180,E1 10059.852,E2 10059.852} C_VEL
LIN {X 0,Y 366.599,Z 930.979,A -85,B 0,C 180,E1 10056.193,E2 10056.193} C_VEL
LIN {X 0,Y 362.94,Z 955.721,A -85,B 0,C 180,E1 10055.601,E2 10055.601} C_VEL
LIN {X 0,Y 358.723,Z 976.776,A -85,B 0,C 180,E1 10054.928,E2 10054.928} C_VEL
LIN {X 0,Y 353.027,Z 999.177,A -85,B 0,C 180,E1 10054.002,E2 10054.002} C_VEL
LIN {X 0,Y 346.618,Z 1020.23,A -85,B 0,C 180,E1 10052.91,E2 10052.91} C_VEL
LIN {X 0,Y 338.596,Z 1042.511,A -85,B 0,C 180,E1 10051.462,E2 10051.462} C_VEL
LIN {X 0,Y 330.085,Z 1063.267,A -85,B 0,C 180,E1 10049.811,E2 10049.811} C_VEL
LIN {X 0,Y 320.687,Z 1083.289,A -85,B 0,C 180,E1 10047.833,E2 10047.833} C_VEL
LIN {X 0,Y 310.637,Z 1102.777,A -85,B 0,C 180,E1 10045.487,E2 10045.487} C_VEL
LIN {X 0,Y 301.1,Z 1119.641,A -85,B 0,C 180,E1 10042.999,E2 10042.999} C_VEL
LIN {X 0,Y 290.465,Z 1137.182,A -85,B 0,C 180,E1 10039.834,E2 10039.834} C_VEL
LIN {X 0,Y 281.342,Z 1151.422,A -85,B 0,C 180,E1 10036.692,E2 10036.692} C_VEL
LIN {X 0,Y 271.906,Z 1165.568,A -85,B 0,C 180,E1 10032.866,E2 10032.866} C_VEL
LIN {X 0,Y 263.943,Z 1177.344,A -85,B 0,C 180,E1 10028.964,E2 10028.964} C_VEL
LIN {X 0,Y 256.151,Z 1188.926,A -85,B 0,C 180,E1 10024.2,E2 10024.2} C_VEL
LIN {X 0,Y 250.144,Z 1198.35,A -85,B 0,C 180,E1 10019.378,E2 10019.378} C_VEL
LIN {X 0,Y 245.364,Z 1206.467,A -85,B 0,C 180,E1 10014.048,E2 10014.048} C_VEL
LIN {X 0,Y 242.312,Z 1212.743,A -85,B 0,C 180,E1 10008.775,E2 10008.775} C_VEL
LIN {X 0,Y 240.623,Z 1217.313,A -85,B 0,C 180,E1 10003.456,E2 10003.456} C_VEL
LIN {X 0,Y 240.059,Z 1220.07,A -85,B 0,C 180,E1 9998.865,E2 9998.865} C_VEL
LIN {X 0,Y 239.972,Z 1221.808,A -85,B 0,C 180,E1 9994.062,E2 9994.062} C_VEL
LIN {X 0,Y 239.995,Z 1222.214,A -85,B 0,C 180,E1 9989.284,E2 9989.284} C_VEL
LIN {X 0,Y 239.956,Z 1221.505,A -85,B 0,C 180,E1 9984.98,E2 9984.98} C_VEL
LIN {X 0,Y 240.088,Z 1219.804,A -85,B 0,C 180,E1 9980.653,E2 9980.653} C_VEL
LIN {X 0,Y 240.903,Z 1216.435,A -85,B 0,C 180,E1 9975.334,E2 9975.334} C_VEL
LIN {X 0,Y 242.874,Z 1211.359,A -85,B 0,C 180,E1 9970.02,E2 9970.02} C_VEL
LIN {X 0,Y 246.263,Z 1204.82,A -85,B 0,C 180,E1 9964.766,E2 9964.766} C_VEL
LIN {X 0,Y 251.219,Z 1196.469,A -85,B 0,C 180,E1 9959.638,E2 9959.638} C_VEL
LIN {X 0,Y 257.783,Z 1186.453,A -85,B 0,C 180,E1 9954.695,E2 9954.695} C_VEL
LIN {X 0,Y 265.511,Z 1174.856,A -85,B 0,C 180,E1 9950.194,E2 9950.194} C_VEL
LIN {X 0,Y 274.186,Z 1162.098,A -85,B 0,C 180,E1 9946.143,E2 9946.143} C_VEL
LIN {X 0,Y 282.972,Z 1148.682,A -85,B 0,C 180,E1 9942.697,E2 9942.697} C_VEL
LIN {X 0,Y 292.71,Z 1133.42,A -85,B 0,C 180,E1 9939.448,E2 9939.448} C_VEL
LIN {X 0,Y 302.575,Z 1116.814,A -85,B 0,C 180,E1 9936.583,E2 9936.583} C_VEL
LIN {X 0,Y 312.837,Z 1098.347,A -85,B 0,C 180,E1 9933.964,E2 9933.964} C_VEL
LIN {X 0,Y 322.038,Z 1080.157,A -85,B 0,C 180,E1 9931.859,E2 9931.859} C_VEL
LIN {X 0,Y 331.535,Z 1059.344,A -85,B 0,C 180,E1 9929.882,E2 9929.882} C_VEL
LIN {X 0,Y 339.284,Z 1040.247,A -85,B 0,C 180,E1 9928.398,E2 9928.398} C_VEL
LIN {X 0,Y 347.215,Z 1017.698,A -85,B 0,C 180,E1 9926.969,E2 9926.969} C_VEL
LIN {X 0,Y 353.477,Z 996.856,A -85,B 0,C 180,E1 9925.907,E2 9925.907} C_VEL
LIN {X 0,Y 359.232,Z 973.375,A -85,B 0,C 180,E1 9924.971,E2 9924.971} C_VEL
LIN {X 0,Y 363.475,Z 951.616,A -85,B 0,C 180,E1 9924.303,E2 9924.303} C_VEL
LIN {X 0,Y 366.732,Z 927.677,A -85,B 0,C 180,E1 9923.761,E2 9923.761} C_VEL
LIN {X 0,Y 385.337,Z 718.391,A -85,B 0,C 180,E1 9920.149,E2 9920.149} C_VEL
LIN {X 0,Y 379.724,Z 708.515,A -85,B 0,C 180,E1 9917.587,E2 9917.587} C_VEL
LIN {X 0,Y 374.343,Z 699.75,A -85,B 0,C 180,E1 9914.779,E2 9914.779} C_VEL
LIN {X 0,Y 370.057,Z 693.33,A -85,B 0,C 180,E1 9912.167,E2 9912.167} C_VEL
LIN {X 0,Y 367.476,Z 689.662,A -85,B 0,C 180,E1 9910.346,E2 9910.346} C_VEL
LIN {X 0,Y 365.209,Z 686.492,A -85,B 0,C 180,E1 9908.502,E2 9908.502} C_VEL
LIN {X 0,Y 362.262,Z 682.554,A -85,B 0,C 180,E1 9905.544,E2 9905.544} C_VEL
LIN {X 0,Y 359.276,Z 679.682,A -85,B 0,C 180,E1 9900.957,E2 9900.957} C_VEL
LIN {X 0,Y 358.341,Z 679.468,A -85,B 0,C 180,E1 9897.761,E2 9897.761} C_VEL
LIN {X 0,Y 358.73,Z 681.456,A -85,B 0,C 180,E1 9892.955,E2 9892.955} C_VEL
LIN {X 0,Y 360.465,Z 685.915,A -85,B 0,C 180,E1 9889.208,E2 9889.208} C_VEL
LIN {X 0,Y 362.843,Z 690.775,A -85,B 0,C 180,E1 9886.21,E2 9886.21} C_VEL
LIN {X 0,Y 366.87,Z 699.07,A -85,B 0,C 180,E1 9882.554,E2 9882.554} C_VEL
LIN {X 0,Y 371.093,Z 707.953,A -85,B 0,C 180,E1 9879.578,E2 9879.578} C_VEL
LIN {X 0,Y 375.35,Z 717.071,A -85,B 0,C 180,E1 9877.071,E2 9877.071} C_VEL
LIN {X 0,Y 380.371,Z 728.361,A -85,B 0,C 180,E1 9874.503,E2 9874.503} C_VEL
LIN {X 0,Y 381.915,Z 732.297,A -85,B 0,C 180,E1 9873.76,E2 9873.76} C_VEL
LIN {X 0,Y 382.041,Z 743.099,A -85,B 0,C 180,E1 9873.229,E2 9873.229} C_VEL
LIN {X 0,Y 365.653,Z 943.563,A -85,B 0,C 180,E1 9869.972,E2 9869.972} C_VEL
LIN {X 0,Y 362.223,Z 966.808,A -85,B 0,C 180,E1 9869.454,E2 9869.454} C_VEL
LIN {X 0,Y 357.642,Z 988.872,A -85,B 0,C 180,E1 9868.813,E2 9868.813} C_VEL
LIN {X 0,Y 351.986,Z 1009.835,A -85,B 0,C 180,E1 9867.986,E2 9867.986} C_VEL
LIN {X 0,Y 344.989,Z 1031.516,A -85,B 0,C 180,E1 9866.886,E2 9866.886} C_VEL
LIN {X 0,Y 337.786,Z 1050.422,A -85,B 0,C 180,E1 9865.675,E2 9865.675} C_VEL
LIN {X 0,Y 328.692,Z 1071.177,A -85,B 0,C 180,E1 9864.013,E2 9864.013} C_VEL
LIN {X 0,Y 319.549,Z 1089.729,A -85,B 0,C 180,E1 9862.171,E2 9862.171} C_VEL
LIN {X 0,Y 309.896,Z 1107.074,A -85,B 0,C 180,E1 9860.021,E2 9860.021} C_VEL
LIN {X 0,Y 299.814,Z 1123.755,A -85,B 0,C 180,E1 9857.478,E2 9857.478} C_VEL
LIN {X 0,Y 290.088,Z 1138.544,A -85,B 0,C 180,E1 9854.679,E2 9854.679} C_VEL
LIN {X 0,Y 280.098,Z 1152.771,A -85,B 0,C 180,E1 9851.329,E2 9851.329} C_VEL
LIN {X 0,Y 271.117,Z 1165.026,A -85,B 0,C 180,E1 9847.748,E2 9847.748} C_VEL
LIN {X 0,Y 262.837,Z 1175.842,A -85,B 0,C 180,E1 9843.738,E2 9843.738} C_VEL
LIN {X 0,Y 255.365,Z 1185.646,A -85,B 0,C 180,E1 9839.171,E2 9839.171} C_VEL
LIN {X 0,Y 249.686,Z 1193.212,A -85,B 0,C 180,E1 9834.612,E2 9834.612} C_VEL
LIN {X 0,Y 244.839,Z 1200.175,A -85,B 0,C 180,E1 9829.068,E2 9829.068} C_VEL
LIN {X 0,Y 241.941,Z 1205.1,A -85,B 0,C 180,E1 9823.625,E2 9823.625} C_VEL
LIN {X 0,Y 240.527,Z 1208.098,A -85,B 0,C 180,E1 9818.354,E2 9818.354} C_VEL
LIN {X 0,Y 240.072,Z 1209.734,A -85,B 0,C 180,E1 9813.104,E2 9813.104} C_VEL
LIN {X 0,Y 240.033,Z 1209.895,A -85,B 0,C 180,E1 9808.568,E2 9808.568} C_VEL
LIN {X 0,Y 240.227,Z 1209.052,A -85,B 0,C 180,E1 9804.027,E2 9804.027} C_VEL
LIN {X 0,Y 241.2,Z 1206.561,A -85,B 0,C 180,E1 9798.523,E2 9798.523} C_VEL
LIN {X 0,Y 243.205,Z 1202.861,A -85,B 0,C 180,E1 9793.521,E2 9793.521} C_VEL
LIN {X 0,Y 246.955,Z 1197.112,A -85,B 0,C 180,E1 9788.131,E2 9788.131} C_VEL
LIN {X 0,Y 252.198,Z 1189.985,A -85,B 0,C 180,E1 9783.131,E2 9783.131} C_VEL
LIN {X 0,Y 258.717,Z 1181.334,A -85,B 0,C 180,E1 9778.552,E2 9778.552} C_VEL
LIN {X 0,Y 267.106,Z 1170.406,A -85,B 0,C 180,E1 9774.006,E2 9774.006} C_VEL
LIN {X 0,Y 275.782,Z 1158.902,A -85,B 0,C 180,E1 9770.232,E2 9770.232} C_VEL
LIN {X 0,Y 285.085,Z 1145.962,A -85,B 0,C 180,E1 9766.847,E2 9766.847} C_VEL
LIN {X 0,Y 294.996,Z 1131.531,A -85,B 0,C 180,E1 9763.785,E2 9763.785} C_VEL
LIN {X 0,Y 305.071,Z 1115.514,A -85,B 0,C 180,E1 9761.078,E2 9761.078} C_VEL
LIN {X 0,Y 315.337,Z 1097.795,A -85,B 0,C 180,E1 9758.657,E2 9758.657} C_VEL
LIN {X 0,Y 324.426,Z 1080.485,A -85,B 0,C 180,E1 9756.746,E2 9756.746} C_VEL
LIN {X 0,Y 333.359,Z 1061.319,A -85,B 0,C 180,E1 9755.033,E2 9755.033} C_VEL
LIN {X 0,Y 341.712,Z 1041.095,A -85,B 0,C 180,E1 9753.576,E2 9753.576} C_VEL
LIN {X 0,Y 348.924,Z 1020.421,A -85,B 0,C 180,E1 9752.403,E2 9752.403} C_VEL
LIN {X 0,Y 355.73,Z 997.13,A -85,B 0,C 180,E1 9751.378,E2 9751.378} C_VEL
LIN {X 0,Y 360.858,Z 975.332,A -85,B 0,C 180,E1 9750.659,E2 9750.659} C_VEL
LIN {X 0,Y 364.728,Z 952.498,A -85,B 0,C 180,E1 9750.104,E2 9750.104} C_VEL
LIN {X 0,Y 367.413,Z 927.02,A -85,B 0,C 180,E1 9749.628,E2 9749.628} C_VEL
LIN {X 0,Y 382.334,Z 741.198,A -85,B 0,C 180,E1 9746.602,E2 9746.602} C_VEL
LIN {X 0,Y 382.042,Z 732.004,A -85,B 0,C 180,E1 9746.085,E2 9746.085} C_VEL
LIN {X 0,Y 377.326,Z 721.112,A -85,B 0,C 180,E1 9743.753,E2 9743.753} C_VEL
LIN {X 0,Y 372.434,Z 710.53,A -85,B 0,C 180,E1 9741.003,E2 9741.003} C_VEL
LIN {X 0,Y 368.562,Z 702.323,A -85,B 0,C 180,E1 9738.425,E2 9738.425} C_VEL
LIN {X 0,Y 366.559,Z 698.136,A -85,B 0,C 180,E1 9736.887,E2 9736.887} C_VEL
LIN {X 0,Y 365.054,Z 696.492,A -85,B 0,C 180,E1 9735.722,E2 9735.722} C_VEL
LIN {X 0,Y 362.129,Z 696.37,A -85,B 0,C 180,E1 9733.38,E2 9733.38} C_VEL
LIN {X 0,Y 360.496,Z 695.797,A -85,B 0,C 180,E1 9731.708,E2 9731.708} C_VEL
LIN {X 0,Y 360.234,Z 695.367,A -85,B 0,C 180,E1 9731.36,E2 9731.36} C_VEL
LIN {X 0,Y 359.003,Z 692.477,A -85,B 0,C 180,E1 9729.296,E2 9729.296} C_VEL
LIN {X 0,Y 357.851,Z 689.064,A -85,B 0,C 180,E1 9725.934,E2 9725.934} C_VEL
LIN {X 0,Y 357.901,Z 687.709,A -85,B 0,C 180,E1 9721.121,E2 9721.121} C_VEL
LIN {X 0,Y 359.145,Z 688.488,A -85,B 0,C 180,E1 9717.926,E2 9717.926} C_VEL
LIN {X 0,Y 361.758,Z 691.197,A -85,B 0,C 180,E1 9714.21,E2 9714.21} C_VEL
LIN {X 0,Y 365.098,Z 695.802,A -85,B 0,C 180,E1 9710.94,E2 9710.94} C_VEL
LIN {X 0,Y 368.183,Z 700.266,A -85,B 0,C 180,E1 9708.565,E2 9708.565} C_VEL
LIN {X 0,Y 372.45,Z 706.788,A -85,B 0,C 180,E1 9705.82,E2 9705.82} C_VEL
LIN {X 0,Y 377.627,Z 715.465,A -85,B 0,C 180,E1 9702.987,E2 9702.987} C_VEL
LIN {X 0,Y 382.021,Z 723.285,A -85,B 0,C 180,E1 9700.88,E2 9700.88} C_VEL
LIN {X 0,Y 363.051,Z 931.171,A -85,B 0,C 180,E1 9697.32,E2 9697.32} C_VEL
LIN {X 0,Y 359.312,Z 955.987,A -85,B 0,C 180,E1 9696.733,E2 9696.733} C_VEL
LIN {X 0,Y 355.008,Z 977.056,A -85,B 0,C 180,E1 9696.067,E2 9696.067} C_VEL
LIN {X 0,Y 349.258,Z 999.209,A -85,B 0,C 180,E1 9695.163,E2 9695.163} C_VEL
LIN {X 0,Y 342.87,Z 1019.785,A -85,B 0,C 180,E1 9694.109,E2 9694.109} C_VEL
LIN {X 0,Y 334.645,Z 1042.222,A -85,B 0,C 180,E1 9692.673,E2 9692.673} C_VEL
LIN {X 0,Y 326.134,Z 1062.522,A -85,B 0,C 180,E1 9691.078,E2 9691.078} C_VEL
LIN {X 0,Y 316.725,Z 1082.186,A -85,B 0,C 180,E1 9689.167,E2 9689.167} C_VEL
LIN {X 0,Y 306.693,Z 1101.29,A -85,B 0,C 180,E1 9686.914,E2 9686.914} C_VEL
LIN {X 0,Y 296.504,Z 1118.793,A -85,B 0,C 180,E1 9684.359,E2 9684.359} C_VEL
LIN {X 0,Y 285.764,Z 1136.028,A -85,B 0,C 180,E1 9681.284,E2 9681.284} C_VEL
LIN {X 0,Y 276.367,Z 1150.161,A -85,B 0,C 180,E1 9678.183,E2 9678.183} C_VEL
LIN {X 0,Y 265.882,Z 1165.314,A -85,B 0,C 180,E1 9674.083,E2 9674.083} C_VEL
LIN {X 0,Y 257.449,Z 1177.221,A -85,B 0,C 180,E1 9670.082,E2 9670.082} C_VEL
LIN {X 0,Y 249.329,Z 1188.697,A -85,B 0,C 180,E1 9665.273,E2 9665.273} C_VEL
LIN {X 0,Y 243.033,Z 1198.011,A -85,B 0,C 180,E1 9660.4,E2 9660.4} C_VEL
LIN {X 0,Y 237.853,Z 1206.249,A -85,B 0,C 180,E1 9654.858,E2 9654.858} C_VEL
LIN {X 0,Y 234.558,Z 1212.528,A -85,B 0,C 180,E1 9649.42,E2 9649.42} C_VEL
LIN {X 0,Y 232.684,Z 1217.193,A -85,B 0,C 180,E1 9643.791,E2 9643.791} C_VEL
LIN {X 0,Y 232.062,Z 1219.983,A -85,B 0,C 180,E1 9638.923,E2 9638.923} C_VEL
LIN {X 0,Y 231.974,Z 1221.674,A -85,B 0,C 180,E1 9633.954,E2 9633.954} C_VEL
LIN {X 0,Y 231.998,Z 1222.004,A -85,B 0,C 180,E1 9629.204,E2 9629.204} C_VEL
LIN {X 0,Y 231.958,Z 1221.275,A -85,B 0,C 180,E1 9624.725,E2 9624.725} C_VEL
LIN {X 0,Y 232.107,Z 1219.596,A -85,B 0,C 180,E1 9620.328,E2 9620.328} C_VEL
LIN {X 0,Y 233.021,Z 1216.225,A -85,B 0,C 180,E1 9614.827,E2 9614.827} C_VEL
LIN {X 0,Y 235.201,Z 1211.076,A -85,B 0,C 180,E1 9609.272,E2 9609.272} C_VEL
LIN {X 0,Y 238.819,Z 1204.601,A -85,B 0,C 180,E1 9603.922,E2 9603.922} C_VEL
LIN {X 0,Y 244.103,Z 1196.24,A -85,B 0,C 180,E1 9598.654,E2 9598.654} C_VEL
LIN {X 0,Y 250.697,Z 1186.7,A -85,B 0,C 180,E1 9593.824,E2 9593.824} C_VEL
LIN {X 0,Y 258.762,Z 1175.201,A -85,B 0,C 180,E1 9589.231,E2 9589.231} C_VEL
LIN {X 0,Y 267.778,Z 1162.544,A -85,B 0,C 180,E1 9585.113,E2 9585.113} C_VEL
LIN {X 0,Y 277.411,Z 1148.4,A -85,B 0,C 180,E1 9581.437,E2 9581.437} C_VEL
LIN {X 0,Y 287.769,Z 1132.691,A -85,B 0,C 180,E1 9578.096,E2 9578.096} C_VEL
LIN {X 0,Y 297.726,Z 1116.478,A -85,B 0,C 180,E1 9575.307,E2 9575.307} C_VEL
LIN {X 0,Y 308.639,Z 1097.331,A -85,B 0,C 180,E1 9572.618,E2 9572.618} C_VEL
LIN {X 0,Y 317.733,Z 1079.813,A -85,B 0,C 180,E1 9570.609,E2 9570.609} C_VEL
LIN {X 0,Y 327.51,Z 1058.855,A -85,B 0,C 180,E1 9568.641,E2 9568.641} C_VEL
LIN {X 0,Y 335.886,Z 1038.621,A -85,B 0,C 180,E1 9567.095,E2 9567.095} C_VEL
LIN {X 0,Y 343.584,Z 1016.931,A -85,B 0,C 180,E1 9565.754,E2 9565.754} C_VEL
LIN {X 0,Y 350.404,Z 994.52,A -85,B 0,C 180,E1 9564.638,E2 9564.638} C_VEL
LIN {X 0,Y 356.024,Z 971.341,A -85,B 0,C 180,E1 9563.752,E2 9563.752} C_VEL
LIN {X 0,Y 360.545,Z 947.585,A -85,B 0,C 180,E1 9563.061,E2 9563.061} C_VEL
LIN {X 0,Y 363.513,Z 924.849,A -85,B 0,C 180,E1 9562.577,E2 9562.577} C_VEL
LIN {X 0,Y 381.762,Z 722.987,A -85,B 0,C 180,E1 9559.111,E2 9559.111} C_VEL
LIN {X 0,Y 375.854,Z 712.56,A -85,B 0,C 180,E1 9556.22,E2 9556.22} C_VEL
LIN {X 0,Y 370.789,Z 704.368,A -85,B 0,C 180,E1 9553.33,E2 9553.33} C_VEL
LIN {X 0,Y 366.569,Z 697.991,A -85,B 0,C 180,E1 9550.451,E2 9550.451} C_VEL
LIN {X 0,Y 363.852,Z 694.18,A -85,B 0,C 180,E1 9548.216,E2 9548.216} C_VEL
LIN {X 0,Y 360.995,Z 690.326,A -85,B 0,C 180,E1 9545.244,E2 9545.244} C_VEL
LIN {X 0,Y 358.221,Z 687.576,A -85,B 0,C 180,E1 9540.8,E2 9540.8} C_VEL
LIN {X 0,Y 357.342,Z 687.455,A -85,B 0,C 180,E1 9537.594,E2 9537.594} C_VEL
LIN {X 0,Y 357.707,Z 689.364,A -85,B 0,C 180,E1 9533.096,E2 9533.096} C_VEL
LIN {X 0,Y 359.341,Z 693.747,A -85,B 0,C 180,E1 9529.418,E2 9529.418} C_VEL
LIN {X 0,Y 361.577,Z 698.484,A -85,B 0,C 180,E1 9526.486,E2 9526.486} C_VEL
LIN {X 0,Y 365.341,Z 706.572,A -85,B 0,C 180,E1 9522.931,E2 9522.931} C_VEL
LIN {X 0,Y 369.275,Z 715.128,A -85,B 0,C 180,E1 9520.052,E2 9520.052} C_VEL
LIN {X 0,Y 373.599,Z 724.663,A -85,B 0,C 180,E1 9517.416,E2 9517.416} C_VEL
LIN {X 0,Y 378.651,Z 736.517,A -85,B 0,C 180,E1 9514.756,E2 9514.756} C_VEL
LIN {X 0,Y 378.807,Z 738.563,A -85,B 0,C 180,E1 9514.6,E2 9514.6} C_VEL
LIN {X 0,Y 378.791,Z 744.654,A -85,B 0,C 180,E1 9514.316,E2 9514.316} C_VEL
LIN {X 0,Y 362.087,Z 943.422,A -85,B 0,C 180,E1 9511.103,E2 9511.103} C_VEL
LIN {X 0,Y 358.578,Z 966.667,A -85,B 0,C 180,E1 9510.59,E2 9510.59} C_VEL
LIN {X 0,Y 353.982,Z 988.439,A -85,B 0,C 180,E1 9509.967,E2 9509.967} C_VEL
LIN {X 0,Y 348.214,Z 1009.433,A -85,B 0,C 180,E1 9509.153,E2 9509.153} C_VEL
LIN {X 0,Y 341.445,Z 1030.173,A -85,B 0,C 180,E1 9508.126,E2 9508.126} C_VEL
LIN {X 0,Y 334.075,Z 1049.211,A -85,B 0,C 180,E1 9506.931,E2 9506.931} C_VEL
LIN {X 0,Y 325.112,Z 1069.454,A -85,B 0,C 180,E1 9505.353,E2 9505.353} C_VEL
LIN {X 0,Y 316.095,Z 1087.419,A -85,B 0,C 180,E1 9503.612,E2 9503.612} C_VEL
LIN {X 0,Y 306.09,Z 1105.232,A -85,B 0,C 180,E1 9501.475,E2 9501.475} C_VEL
LIN {X 0,Y 296.169,Z 1121.427,A -85,B 0,C 180,E1 9499.083,E2 9499.083} C_VEL
LIN {X 0,Y 286.115,Z 1136.337,A -85,B 0,C 180,E1 9496.334,E2 9496.334} C_VEL
LIN {X 0,Y 276.171,Z 1150.281,A -85,B 0,C 180,E1 9493.178,E2 9493.178} C_VEL
LIN {X 0,Y 266.628,Z 1162.79,A -85,B 0,C 180,E1 9489.606,E2 9489.606} C_VEL
LIN {X 0,Y 256.933,Z 1175.071,A -85,B 0,C 180,E1 9485.166,E2 9485.166} C_VEL
LIN {X 0,Y 249.143,Z 1184.866,A -85,B 0,C 180,E1 9480.642,E2 9480.642} C_VEL
LIN {X 0,Y 242.589,Z 1193.088,A -85,B 0,C 180,E1 9475.643,E2 9475.643} C_VEL
LIN {X 0,Y 237.372,Z 1200.141,A -85,B 0,C 180,E1 9469.949,E2 9469.949} C_VEL
LIN {X 0,Y 234.299,Z 1204.931,A -85,B 0,C 180,E1 9464.583,E2 9464.583} C_VEL
LIN {X 0,Y 232.666,Z 1208.082,A -85,B 0,C 180,E1 9459.149,E2 9459.149} C_VEL
LIN {X 0,Y 232.118,Z 1209.733,A -85,B 0,C 180,E1 9454.199,E2 9454.199} C_VEL
LIN {X 0,Y 232.036,Z 1210.143,A -85,B 0,C 180,E1 9449.012,E2 9449.012} C_VEL
LIN {X 0,Y 232.205,Z 1209.385,A -85,B 0,C 180,E1 9444.316,E2 9444.316} C_VEL
LIN {X 0,Y 233.102,Z 1207.225,A -85,B 0,C 180,E1 9438.871,E2 9438.871} C_VEL
LIN {X 0,Y 235.19,Z 1203.464,A -85,B 0,C 180,E1 9433.451,E2 9433.451} C_VEL
LIN {X 0,Y 239.235,Z 1197.616,A -85,B 0,C 180,E1 9427.646,E2 9427.646} C_VEL
LIN {X 0,Y 244.795,Z 1190.432,A -85,B 0,C 180,E1 9422.42,E2 9422.42} C_VEL
LIN {X 0,Y 251.825,Z 1181.554,A -85,B 0,C 180,E1 9417.588,E2 9417.588} C_VEL
LIN {X 0,Y 260.155,Z 1171.197,A -85,B 0,C 180,E1 9413.162,E2 9413.162} C_VEL
LIN {X 0,Y 268.898,Z 1160.034,A -85,B 0,C 180,E1 9409.405,E2 9409.405} C_VEL
LIN {X 0,Y 279.233,Z 1146.233,A -85,B 0,C 180,E1 9405.714,E2 9405.714} C_VEL
LIN {X 0,Y 289.47,Z 1131.814,A -85,B 0,C 180,E1 9402.632,E2 9402.632} C_VEL
LIN {X 0,Y 299.841,Z 1115.826,A -85,B 0,C 180,E1 9399.918,E2 9399.918} C_VEL
LIN {X 0,Y 310.283,Z 1098.346,A -85,B 0,C 180,E1 9397.521,E2 9397.521} C_VEL
LIN {X 0,Y 319.694,Z 1080.887,A -85,B 0,C 180,E1 9395.594,E2 9395.594} C_VEL
LIN {X 0,Y 328.833,Z 1061.816,A -85,B 0,C 180,E1 9393.892,E2 9393.892} C_VEL
LIN {X 0,Y 337.224,Z 1042.049,A -85,B 0,C 180,E1 9392.469,E2 9392.469} C_VEL
LIN {X 0,Y 344.655,Z 1021.357,A -85,B 0,C 180,E1 9391.296,E2 9391.296} C_VEL
LIN {X 0,Y 351.277,Z 999.635,A -85,B 0,C 180,E1 9390.327,E2 9390.327} C_VEL
LIN {X 0,Y 356.487,Z 978.298,A -85,B 0,C 180,E1 9389.613,E2 9389.613} C_VEL
LIN {X 0,Y 360.858,Z 954.309,A -85,B 0,C 180,E1 9389.014,E2 9389.014} C_VEL
LIN {X 0,Y 363.558,Z 931.1,A -85,B 0,C 180,E1 9388.567,E2 9388.567} C_VEL
LIN {X 0,Y 379.099,Z 742.733,A -85,B 0,C 180,E1 9385.515,E2 9385.515} C_VEL
LIN {X 0,Y 378.916,Z 736.822,A -85,B 0,C 180,E1 9385.166,E2 9385.166} C_VEL
LIN {X 0,Y 373.984,Z 725.16,A -85,B 0,C 180,E1 9382.561,E2 9382.561} C_VEL
LIN {X 0,Y 369.259,Z 714.718,A -85,B 0,C 180,E1 9379.661,E2 9379.661} C_VEL
LIN {X 0,Y 364.921,Z 705.344,A -85,B 0,C 180,E1 9376.393,E2 9376.393} C_VEL
LIN {X 0,Y 361.403,Z 697.769,A -85,B 0,C 180,E1 9372.869,E2 9372.869} C_VEL
LIN {X 0,Y 360.234,Z 695.367,A -85,B 0,C 180,E1 9371.36,E2 9371.36} C_VEL
LIN {X 0,Y 359.337,Z 694.592,A -85,B 0,C 180,E1 9370.142,E2 9370.142} C_VEL
LIN {X 0,Y 357.792,Z 696.013,A -85,B 0,C 180,E1 9367.933,E2 9367.933} C_VEL
LIN {X 0,Y 356.912,Z 697.007,A -85,B 0,C 180,E1 9366.053,E2 9366.053} C_VEL
LIN {X 0,Y 356.82,Z 696.913,A -85,B 0,C 180,E1 9365.693,E2 9365.693} C_VEL
LIN {X 0,Y 357.013,Z 695.629,A -85,B 0,C 180,E1 9360.802,E2 9360.802} C_VEL
LIN {X 0,Y 358.249,Z 696.568,A -85,B 0,C 180,E1 9357.761,E2 9357.761} C_VEL
LIN {X 0,Y 360.561,Z 698.99,A -85,B 0,C 180,E1 9354.43,E2 9354.43} C_VEL
LIN {X 0,Y 363.81,Z 703.622,A -85,B 0,C 180,E1 9351.146,E2 9351.146} C_VEL
LIN {X 0,Y 366.839,Z 708.128,A -85,B 0,C 180,E1 9348.762,E2 9348.762} C_VEL
LIN {X 0,Y 370.839,Z 714.452,A -85,B 0,C 180,E1 9346.115,E2 9346.115} C_VEL
LIN {X 0,Y 375.921,Z 723.182,A -85,B 0,C 180,E1 9343.266,E2 9343.266} C_VEL
LIN {X 0,Y 378.58,Z 728.221,A -85,B 0,C 180,E1 9341.919,E2 9341.919} C_VEL
LIN {X 0,Y 359.616,Z 931.648,A -85,B 0,C 180,E1 9338.463,E2 9338.463} C_VEL
LIN {X 0,Y 355.819,Z 956.301,A -85,B 0,C 180,E1 9337.886,E2 9337.886} C_VEL
LIN {X 0,Y 351.413,Z 977.438,A -85,B 0,C 180,E1 9337.225,E2 9337.225} C_VEL
LIN {X 0,Y 345.521,Z 999.628,A -85,B 0,C 180,E1 9336.33,E2 9336.33} C_VEL
LIN {X 0,Y 338.725,Z 1021.008,A -85,B 0,C 180,E1 9335.242,E2 9335.242} C_VEL
LIN {X 0,Y 330.713,Z 1042.269,A -85,B 0,C 180,E1 9333.887,E2 9333.887} C_VEL
LIN {X 0,Y 321.885,Z 1062.832,A -85,B 0,C 180,E1 9332.286,E2 9332.286} C_VEL
LIN {X 0,Y 312.24,Z 1082.446,A -85,B 0,C 180,E1 9330.389,E2 9330.389} C_VEL
LIN {X 0,Y 301.935,Z 1101.503,A -85,B 0,C 180,E1 9328.146,E2 9328.146} C_VEL
LIN {X 0,Y 291.447,Z 1118.98,A -85,B 0,C 180,E1 9325.596,E2 9325.596} C_VEL
LIN {X 0,Y 280.062,Z 1136.606,A -85,B 0,C 180,E1 9322.426,E2 9322.426} C_VEL
LIN {X 0,Y 269.815,Z 1151.466,A -85,B 0,C 180,E1 9319.11,E2 9319.11} C_VEL
LIN {X 0,Y 259.493,Z 1165.716,A -85,B 0,C 180,E1 9315.151,E2 9315.151} C_VEL
LIN {X 0,Y 250.388,Z 1178.034,A -85,B 0,C 180,E1 9310.911,E2 9310.911} C_VEL
LIN {X 0,Y 242.246,Z 1188.942,A -85,B 0,C 180,E1 9306.173,E2 9306.173} C_VEL
LIN {X 0,Y 235.371,Z 1198.622,A -85,B 0,C 180,E1 9300.931,E2 9300.931} C_VEL
LIN {X 0,Y 230.075,Z 1206.54,A -85,B 0,C 180,E1 9295.317,E2 9295.317} C_VEL
LIN {X 0,Y 226.59,Z 1212.816,A -85,B 0,C 180,E1 9289.594,E2 9289.594} C_VEL
LIN {X 0,Y 224.697,Z 1217.232,A -85,B 0,C 180,E1 9283.904,E2 9283.904} C_VEL
LIN {X 0,Y 224.045,Z 1220.016,A -85,B 0,C 180,E1 9278.727,E2 9278.727} C_VEL
LIN {X 0,Y 223.976,Z 1221.541,A -85,B 0,C 180,E1 9273.583,E2 9273.583} C_VEL
LIN {X 0,Y 224,Z 1221.781,A -85,B 0,C 180,E1 9268.977,E2 9268.977} C_VEL
LIN {X 0,Y 223.96,Z 1221.094,A -85,B 0,C 180,E1 9264.62,E2 9264.62} C_VEL
LIN {X 0,Y 224.134,Z 1219.389,A -85,B 0,C 180,E1 9259.981,E2 9259.981} C_VEL
LIN {X 0,Y 225.153,Z 1216.015,A -85,B 0,C 180,E1 9254.283,E2 9254.283} C_VEL
LIN {X 0,Y 227.493,Z 1210.928,A -85,B 0,C 180,E1 9248.605,E2 9248.605} C_VEL
LIN {X 0,Y 231.429,Z 1204.384,A -85,B 0,C 180,E1 9243.023,E2 9243.023} C_VEL
LIN {X 0,Y 237.062,Z 1196.011,A -85,B 0,C 180,E1 9237.612,E2 9237.612} C_VEL
LIN {X 0,Y 244.139,Z 1186.343,A -85,B 0,C 180,E1 9232.612,E2 9232.612} C_VEL
LIN {X 0,Y 252.529,Z 1174.954,A -85,B 0,C 180,E1 9228,E2 9228} C_VEL
LIN {X 0,Y 261.956,Z 1162.278,A -85,B 0,C 180,E1 9223.831,E2 9223.831} C_VEL
LIN {X 0,Y 271.993,Z 1148.119,A -85,B 0,C 180,E1 9220.127,E2 9220.127} C_VEL
LIN {X 0,Y 283.039,Z 1131.902,A -85,B 0,C 180,E1 9216.689,E2 9216.689} C_VEL
LIN {X 0,Y 293.031,Z 1116.144,A -85,B 0,C 180,E1 9213.989,E2 9213.989} C_VEL
LIN {X 0,Y 304.279,Z 1096.939,A -85,B 0,C 180,E1 9211.312,E2 9211.312} C_VEL
LIN {X 0,Y 313.986,Z 1078.705,A -85,B 0,C 180,E1 9209.247,E2 9209.247} C_VEL
LIN {X 0,Y 323.678,Z 1058.293,A -85,B 0,C 180,E1 9207.364,E2 9207.364} C_VEL
LIN {X 0,Y 332.189,Z 1038.157,A -85,B 0,C 180,E1 9205.847,E2 9205.847} C_VEL
LIN {X 0,Y 339.73,Z 1017.308,A -85,B 0,C 180,E1 9204.576,E2 9204.576} C_VEL
LIN {X 0,Y 346.653,Z 995.065,A -85,B 0,C 180,E1 9203.478,E2 9203.478} C_VEL
LIN {X 0,Y 352.395,Z 971.948,A -85,B 0,C 180,E1 9202.603,E2 9202.603} C_VEL
LIN {X 0,Y 356.989,Z 948.473,A -85,B 0,C 180,E1 9201.924,E2 9201.924} C_VEL
LIN {X 0,Y 360.054,Z 925.574,A -85,B 0,C 180,E1 9201.44,E2 9201.44} C_VEL
LIN {X 0,Y 378.353,Z 727.812,A -85,B 0,C 180,E1 9198.077,E2 9198.077} C_VEL
LIN {X 0,Y 372.763,Z 717.839,A -85,B 0,C 180,E1 9195.161,E2 9195.161} C_VEL
LIN {X 0,Y 368.015,Z 709.984,A -85,B 0,C 180,E1 9192.235,E2 9192.235} C_VEL
LIN {X 0,Y 364.661,Z 705.004,A -85,B 0,C 180,E1 9189.788,E2 9189.788} C_VEL
LIN {X 0,Y 362.507,Z 701.869,A -85,B 0,C 180,E1 9187.927,E2 9187.927} C_VEL
LIN {X 0,Y 359.876,Z 698.2,A -85,B 0,C 180,E1 9185.101,E2 9185.101} C_VEL
LIN {X 0,Y 357.233,Z 695.524,A -85,B 0,C 180,E1 9180.802,E2 9180.802} C_VEL
LIN {X 0,Y 356.38,Z 695.364,A -85,B 0,C 180,E1 9177.749,E2 9177.749} C_VEL
LIN {X 0,Y 356.694,Z 697.273,A -85,B 0,C 180,E1 9173.239,E2 9173.239} C_VEL
LIN {X 0,Y 358.222,Z 701.577,A -85,B 0,C 180,E1 9169.628,E2 9169.628} C_VEL
LIN {X 0,Y 360.318,Z 706.193,A -85,B 0,C 180,E1 9166.765,E2 9166.765} C_VEL
LIN {X 0,Y 363.88,Z 714.183,A -85,B 0,C 180,E1 9163.271,E2 9163.271} C_VEL
LIN {X 0,Y 367.477,Z 722.3,A -85,B 0,C 180,E1 9160.53,E2 9160.53} C_VEL
LIN {X 0,Y 371.669,Z 731.859,A -85,B 0,C 180,E1 9157.874,E2 9157.874} C_VEL
LIN {X 0,Y 375.741,Z 741.816,A -85,B 0,C 180,E1 9155.617,E2 9155.617} C_VEL
LIN {X 0,Y 375.66,Z 746.365,A -85,B 0,C 180,E1 9155.42,E2 9155.42} C_VEL
LIN {X 0,Y 358.697,Z 942.953,A -85,B 0,C 180,E1 9152.263,E2 9152.263} C_VEL
LIN {X 0,Y 355.117,Z 966.318,A -85,B 0,C 180,E1 9151.754,E2 9151.754} C_VEL
LIN {X 0,Y 350.269,Z 988.747,A -85,B 0,C 180,E1 9151.12,E2 9151.12} C_VEL
LIN {X 0,Y 344.59,Z 1009.031,A -85,B 0,C 180,E1 9150.345,E2 9150.345} C_VEL
LIN {X 0,Y 337.683,Z 1029.824,A -85,B 0,C 180,E1 9149.333,E2 9149.333} C_VEL
LIN {X 0,Y 329.786,Z 1049.781,A -85,B 0,C 180,E1 9148.094,E2 9148.094} C_VEL
LIN {X 0,Y 320.267,Z 1070.635,A -85,B 0,C 180,E1 9146.466,E2 9146.466} C_VEL
LIN {X 0,Y 310.711,Z 1089.15,A -85,B 0,C 180,E1 9144.662,E2 9144.662} C_VEL
LIN {X 0,Y 300.481,Z 1106.673,A -85,B 0,C 180,E1 9142.524,E2 9142.524} C_VEL
LIN {X 0,Y 289.792,Z 1123.439,A -85,B 0,C 180,E1 9139.992,E2 9139.992} C_VEL
LIN {X 0,Y 280.008,Z 1137.449,A -85,B 0,C 180,E1 9137.357,E2 9137.357} C_VEL
LIN {X 0,Y 268.696,Z 1152.589,A -85,B 0,C 180,E1 9133.799,E2 9133.799} C_VEL
LIN {X 0,Y 258.923,Z 1164.965,A -85,B 0,C 180,E1 9130.126,E2 9130.126} C_VEL
LIN {X 0,Y 249.921,Z 1175.8,A -85,B 0,C 180,E1 9126.022,E2 9126.022} C_VEL
LIN {X 0,Y 241.841,Z 1185.489,A -85,B 0,C 180,E1 9121.395,E2 9121.395} C_VEL
LIN {X 0,Y 235.298,Z 1193.305,A -85,B 0,C 180,E1 9116.499,E2 9116.499} C_VEL
LIN {X 0,Y 229.77,Z 1200.352,A -85,B 0,C 180,E1 9110.639,E2 9110.639} C_VEL
LIN {X 0,Y 226.488,Z 1205.141,A -85,B 0,C 180,E1 9105.097,E2 9105.097} C_VEL
LIN {X 0,Y 224.725,Z 1208.288,A -85,B 0,C 180,E1 9099.475,E2 9099.475} C_VEL
LIN {X 0,Y 224.128,Z 1209.938,A -85,B 0,C 180,E1 9094.349,E2 9094.349} C_VEL
LIN {X 0,Y 224.036,Z 1210.369,A -85,B 0,C 180,E1 9089.233,E2 9089.233} C_VEL
LIN {X 0,Y 224.203,Z 1209.654,A -85,B 0,C 180,E1 9084.37,E2 9084.37} C_VEL
LIN {X 0,Y 225.13,Z 1207.583,A -85,B 0,C 180,E1 9078.731,E2 9078.731} C_VEL
LIN {X 0,Y 227.308,Z 1203.869,A -85,B 0,C 180,E1 9073.123,E2 9073.123} C_VEL
LIN {X 0,Y 231.317,Z 1198.412,A -85,B 0,C 180,E1 9067.375,E2 9067.375} C_VEL
LIN {X 0,Y 236.628,Z 1191.791,A -85,B 0,C 180,E1 9062.303,E2 9062.303} C_VEL
LIN {X 0,Y 244.258,Z 1182.667,A -85,B 0,C 180,E1 9057.014,E2 9057.014} C_VEL
LIN {X 0,Y 252.821,Z 1172.547,A -85,B 0,C 180,E1 9052.48,E2 9052.48} C_VEL
LIN {X 0,Y 262.291,Z 1160.895,A -85,B 0,C 180,E1 9048.449,E2 9048.449} C_VEL
LIN {X 0,Y 273.051,Z 1147.105,A -85,B 0,C 180,E1 9044.676,E2 9044.676} C_VEL
LIN {X 0,Y 283.456,Z 1132.922,A -85,B 0,C 180,E1 9041.6,E2 9041.6} C_VEL
LIN {X 0,Y 294.091,Z 1117.136,A -85,B 0,C 180,E1 9038.871,E2 9038.871} C_VEL
LIN {X 0,Y 304.355,Z 1100.667,A -85,B 0,C 180,E1 9036.561,E2 9036.561} C_VEL
LIN {X 0,Y 314.387,Z 1082.608,A -85,B 0,C 180,E1 9034.542,E2 9034.542} C_VEL
LIN {X 0,Y 324.441,Z 1062.312,A -85,B 0,C 180,E1 9032.72,E2 9032.72} C_VEL
LIN {X 0,Y 332.968,Z 1042.695,A -85,B 0,C 180,E1 9031.316,E2 9031.316} C_VEL
LIN {X 0,Y 340.585,Z 1022.09,A -85,B 0,C 180,E1 9030.15,E2 9030.15} C_VEL
LIN {X 0,Y 347.276,Z 1000.867,A -85,B 0,C 180,E1 9029.204,E2 9029.204} C_VEL
LIN {X 0,Y 352.729,Z 979.107,A -85,B 0,C 180,E1 9028.478,E2 9028.478} C_VEL
LIN {X 0,Y 357.36,Z 954.486,A -85,B 0,C 180,E1 9027.866,E2 9027.866} C_VEL
LIN {X 0,Y 360.133,Z 931.457,A -85,B 0,C 180,E1 9027.423,E2 9027.423} C_VEL
LIN {X 0,Y 376.01,Z 744.295,A -85,B 0,C 180,E1 9024.411,E2 9024.411} C_VEL
LIN {X 0,Y 375.943,Z 741.91,A -85,B 0,C 180,E1 9024.263,E2 9024.263} C_VEL
LIN {X 0,Y 371.461,Z 731.1,A -85,B 0,C 180,E1 9021.765,E2 9021.765} C_VEL
LIN {X 0,Y 367.37,Z 721.638,A -85,B 0,C 180,E1 9019.105,E2 9019.105} C_VEL
LIN {X 0,Y 363.308,Z 712.546,A -85,B 0,C 180,E1 9015.893,E2 9015.893} C_VEL
LIN {X 0,Y 360.043,Z 705.18,A -85,B 0,C 180,E1 9012.429,E2 9012.429} C_VEL
LIN {X 0,Y 357.958,Z 700.369,A -85,B 0,C 180,E1 9009.162,E2 9009.162} C_VEL
LIN {X 0,Y 356.841,Z 696.956,A -85,B 0,C 180,E1 9005.79,E2 9005.79} C_VEL
LIN {X 0,Y 356.82,Z 696.913,A -85,B 0,C 180,E1 9005.693,E2 9005.693} C_VEL
LIN {X 0,Y 356.516,Z 697.386,A -85,B 0,C 180,E1 9004.45,E2 9004.45} C_VEL
LIN {X 0,Y 356.083,Z 703.259,A -85,B 0,C 180,E1 9000.781,E2 9000.781} C_VEL
LIN {X 0,Y 356.261,Z 703.668,A -85,B 0,C 180,E1 9000.064,E2 9000.064} C_VEL
LIN {X 0,Y 357.522,Z 704.854,A -85,B 0,C 180,E1 8997.275,E2 8997.275} C_VEL
LIN {X 0,Y 359.429,Z 706.899,A -85,B 0,C 180,E1 8994.573,E2 8994.573} C_VEL
LIN {X 0,Y 362.441,Z 711.295,A -85,B 0,C 180,E1 8991.433,E2 8991.433} C_VEL
LIN {X 0,Y 365.297,Z 715.649,A -85,B 0,C 180,E1 8989.113,E2 8989.113} C_VEL
LIN {X 0,Y 369.123,Z 721.896,A -85,B 0,C 180,E1 8986.489,E2 8986.489} C_VEL
LIN {X 0,Y 374.226,Z 730.89,A -85,B 0,C 180,E1 8983.547,E2 8983.547} C_VEL
LIN {X 0,Y 375.267,Z 733.248,A -85,B 0,C 180,E1 8982.976,E2 8982.976} C_VEL
LIN {X 0,Y 356.354,Z 931.866,A -85,B 0,C 180,E1 8979.633,E2 8979.633} C_VEL
LIN {X 0,Y 352.505,Z 956.458,A -85,B 0,C 180,E1 8979.065,E2 8979.065} C_VEL
LIN {X 0,Y 348.017,Z 977.586,A -85,B 0,C 180,E1 8978.416,E2 8978.416} C_VEL
LIN {X 0,Y 341.931,Z 1000.05,A -85,B 0,C 180,E1 8977.522,E2 8977.522} C_VEL
LIN {X 0,Y 335.276,Z 1020.567,A -85,B 0,C 180,E1 8976.494,E2 8976.494} C_VEL
LIN {X 0,Y 326.895,Z 1042.404,A -85,B 0,C 180,E1 8975.124,E2 8975.124} C_VEL
LIN {X 0,Y 317.782,Z 1063.142,A -85,B 0,C 180,E1 8973.526,E2 8973.526} C_VEL
LIN {X 0,Y 307.901,Z 1082.709,A -85,B 0,C 180,E1 8971.645,E2 8971.645} C_VEL
LIN {X 0,Y 297.322,Z 1101.719,A -85,B 0,C 180,E1 8969.417,E2 8969.417} C_VEL
LIN {X 0,Y 286.532,Z 1119.168,A -85,B 0,C 180,E1 8966.875,E2 8966.875} C_VEL
LIN {X 0,Y 274.477,Z 1137.181,A -85,B 0,C 180,E1 8963.615,E2 8963.615} C_VEL
LIN {X 0,Y 264.456,Z 1151.189,A -85,B 0,C 180,E1 8960.469,E2 8960.469} C_VEL
LIN {X 0,Y 253.707,Z 1165.467,A -85,B 0,C 180,E1 8956.481,E2 8956.481} C_VEL
LIN {X 0,Y 244.076,Z 1177.915,A -85,B 0,C 180,E1 8952.141,E2 8952.141} C_VEL
LIN {X 0,Y 235.593,Z 1188.711,A -85,B 0,C 180,E1 8947.365,E2 8947.365} C_VEL
LIN {X 0,Y 228.301,Z 1198.398,A -85,B 0,C 180,E1 8942,E2 8942} C_VEL
LIN {X 0,Y 222.763,Z 1206.133,A -85,B 0,C 180,E1 8936.382,E2 8936.382} C_VEL
LIN {X 0,Y 219.005,Z 1212.365,A -85,B 0,C 180,E1 8930.581,E2 8930.581} C_VEL
LIN {X 0,Y 216.864,Z 1216.855,A -85,B 0,C 180,E1 8924.689,E2 8924.689} C_VEL
LIN {X 0,Y 216.085,Z 1219.689,A -85,B 0,C 180,E1 8919.32,E2 8919.32} C_VEL
LIN {X 0,Y 215.977,Z 1221.312,A -85,B 0,C 180,E1 8913.982,E2 8913.982} C_VEL
LIN {X 0,Y 216.002,Z 1221.577,A -85,B 0,C 180,E1 8908.939,E2 8908.939} C_VEL
LIN {X 0,Y 215.963,Z 1220.888,A -85,B 0,C 180,E1 8904.421,E2 8904.421} C_VEL
LIN {X 0,Y 216.165,Z 1219.181,A -85,B 0,C 180,E1 8899.607,E2 8899.607} C_VEL
LIN {X 0,Y 217.302,Z 1215.804,A -85,B 0,C 180,E1 8893.7,E2 8893.7} C_VEL
LIN {X 0,Y 219.857,Z 1210.711,A -85,B 0,C 180,E1 8887.823,E2 8887.823} C_VEL
LIN {X 0,Y 224.103,Z 1204.159,A -85,B 0,C 180,E1 8882.059,E2 8882.059} C_VEL
LIN {X 0,Y 230.104,Z 1195.785,A -85,B 0,C 180,E1 8876.506,E2 8876.506} C_VEL
LIN {X 0,Y 237.88,Z 1185.739,A -85,B 0,C 180,E1 8871.224,E2 8871.224} C_VEL
LIN {X 0,Y 246.419,Z 1174.706,A -85,B 0,C 180,E1 8866.707,E2 8866.707} C_VEL
LIN {X 0,Y 256.457,Z 1161.749,A -85,B 0,C 180,E1 8862.416,E2 8862.416} C_VEL
LIN {X 0,Y 266.768,Z 1147.783,A -85,B 0,C 180,E1 8858.752,E2 8858.752} C_VEL
LIN {X 0,Y 278.175,Z 1131.587,A -85,B 0,C 180,E1 8855.322,E2 8855.322} C_VEL
LIN {X 0,Y 288.497,Z 1115.81,A -85,B 0,C 180,E1 8852.63,E2 8852.63} C_VEL
LIN {X 0,Y 300.083,Z 1096.548,A -85,B 0,C 180,E1 8849.968,E2 8849.968} C_VEL
LIN {X 0,Y 309.692,Z 1078.96,A -85,B 0,C 180,E1 8847.993,E2 8847.993} C_VEL
LIN {X 0,Y 319.618,Z 1058.592,A -85,B 0,C 180,E1 8846.128,E2 8846.128} C_VEL
LIN {X 0,Y 327.936,Z 1039.395,A -85,B 0,C 180,E1 8844.69,E2 8844.69} C_VEL
LIN {X 0,Y 336.024,Z 1017.683,A -85,B 0,C 180,E1 8843.371,E2 8843.371} C_VEL
LIN {X 0,Y 342.908,Z 996.053,A -85,B 0,C 180,E1 8842.315,E2 8842.315} C_VEL
LIN {X 0,Y 348.81,Z 972.997,A -85,B 0,C 180,E1 8841.445,E2 8841.445} C_VEL
LIN {X 0,Y 353.479,Z 950.013,A -85,B 0,C 180,E1 8840.781,E2 8840.781} C_VEL
LIN {X 0,Y 356.727,Z 926.422,A -85,B 0,C 180,E1 8840.283,E2 8840.283} C_VEL
LIN {X 0,Y 375.036,Z 732.688,A -85,B 0,C 180,E1 8837.014,E2 8837.014} C_VEL
LIN {X 0,Y 370.172,Z 723.856,A -85,B 0,C 180,E1 8834.309,E2 8834.309} C_VEL
LIN {X 0,Y 365.875,Z 716.71,A -85,B 0,C 180,E1 8831.508,E2 8831.508} C_VEL
LIN {X 0,Y 363.171,Z 712.541,A -85,B 0,C 180,E1 8829.429,E2 8829.429} C_VEL
LIN {X 0,Y 361.075,Z 709.442,A -85,B 0,C 180,E1 8827.546,E2 8827.546} C_VEL
LIN {X 0,Y 358.756,Z 706.073,A -85,B 0,C 180,E1 8824.957,E2 8824.957} C_VEL
LIN {X 0,Y 356.189,Z 703.419,A -85,B 0,C 180,E1 8820.643,E2 8820.643} C_VEL
LIN {X 0,Y 355.376,Z 703.354,A -85,B 0,C 180,E1 8817.581,E2 8817.581} C_VEL
LIN {X 0,Y 355.679,Z 705.181,A -85,B 0,C 180,E1 8813.381,E2 8813.381} C_VEL
LIN {X 0,Y 357.055,Z 709.279,A -85,B 0,C 180,E1 8809.92,E2 8809.92} C_VEL
LIN {X 0,Y 359.059,Z 713.901,A -85,B 0,C 180,E1 8807.046,E2 8807.046} C_VEL
LIN {X 0,Y 362.39,Z 721.681,A -85,B 0,C 180,E1 8803.654,E2 8803.654} C_VEL
LIN {X 0,Y 365.703,Z 729.472,A -85,B 0,C 180,E1 8801.012,E2 8801.012} C_VEL
LIN {X 0,Y 369.697,Z 738.914,A -85,B 0,C 180,E1 8798.376,E2 8798.376} C_VEL
LIN {X 0,Y 372.778,Z 746.931,A -85,B 0,C 180,E1 8796.559,E2 8796.559} C_VEL
LIN {X 0,Y 355.437,Z 942.683,A -85,B 0,C 180,E1 8793.44,E2 8793.44} C_VEL
LIN {X 0,Y 351.801,Z 965.982,A -85,B 0,C 180,E1 8792.939,E2 8792.939} C_VEL
LIN {X 0,Y 346.903,Z 988.313,A -85,B 0,C 180,E1 8792.321,E2 8792.321} C_VEL
LIN {X 0,Y 340.723,Z 1009.905,A -85,B 0,C 180,E1 8791.508,E2 8791.508} C_VEL
LIN {X 0,Y 333.068,Z 1032.065,A -85,B 0,C 180,E1 8790.421,E2 8790.421} C_VEL
LIN {X 0,Y 325.262,Z 1051.232,A -85,B 0,C 180,E1 8789.227,E2 8789.227} C_VEL
LIN {X 0,Y 315.916,Z 1071.086,A -85,B 0,C 180,E1 8787.676,E2 8787.676} C_VEL
LIN {X 0,Y 306.142,Z 1089.559,A -85,B 0,C 180,E1 8785.886,E2 8785.886} C_VEL
LIN {X 0,Y 295.658,Z 1107.016,A -85,B 0,C 180,E1 8783.761,E2 8783.761} C_VEL
LIN {X 0,Y 284.678,Z 1123.737,A -85,B 0,C 180,E1 8781.235,E2 8781.235} C_VEL
LIN {X 0,Y 273.995,Z 1138.563,A -85,B 0,C 180,E1 8778.424,E2 8778.424} C_VEL
LIN {X 0,Y 262.915,Z 1152.844,A -85,B 0,C 180,E1 8775.02,E2 8775.02} C_VEL
LIN {X 0,Y 252.537,Z 1165.514,A -85,B 0,C 180,E1 8771.211,E2 8771.211} C_VEL
LIN {X 0,Y 242.968,Z 1176.529,A -85,B 0,C 180,E1 8766.928,E2 8766.928} C_VEL
LIN {X 0,Y 234.22,Z 1186.492,A -85,B 0,C 180,E1 8761.961,E2 8761.961} C_VEL
LIN {X 0,Y 227.493,Z 1194.204,A -85,B 0,C 180,E1 8756.917,E2 8756.917} C_VEL
LIN {X 0,Y 222.006,Z 1200.808,A -85,B 0,C 180,E1 8751.119,E2 8751.119} C_VEL
LIN {X 0,Y 218.459,Z 1205.721,A -85,B 0,C 180,E1 8745.122,E2 8745.122} C_VEL
LIN {X 0,Y 216.686,Z 1208.711,A -85,B 0,C 180,E1 8739.294,E2 8739.294} C_VEL
LIN {X 0,Y 216.09,Z 1210.348,A -85,B 0,C 180,E1 8733.449,E2 8733.449} C_VEL
LIN {X 0,Y 216.044,Z 1210.508,A -85,B 0,C 180,E1 8728.409,E2 8728.409} C_VEL
LIN {X 0,Y 216.268,Z 1209.73,A -85,B 0,C 180,E1 8723.63,E2 8723.63} C_VEL
LIN {X 0,Y 217.453,Z 1207.334,A -85,B 0,C 180,E1 8717.52,E2 8717.52} C_VEL
LIN {X 0,Y 219.982,Z 1203.538,A -85,B 0,C 180,E1 8711.801,E2 8711.801} C_VEL
LIN {X 0,Y 224.549,Z 1197.745,A -85,B 0,C 180,E1 8705.817,E2 8705.817} C_VEL
LIN {X 0,Y 230.726,Z 1190.631,A -85,B 0,C 180,E1 8700.395,E2 8700.395} C_VEL
LIN {X 0,Y 238.67,Z 1181.55,A -85,B 0,C 180,E1 8695.268,E2 8695.268} C_VEL
LIN {X 0,Y 248.3,Z 1170.547,A -85,B 0,C 180,E1 8690.488,E2 8690.488} C_VEL
LIN {X 0,Y 258.401,Z 1158.646,A -85,B 0,C 180,E1 8686.469,E2 8686.469} C_VEL
LIN {X 0,Y 269.064,Z 1145.244,A -85,B 0,C 180,E1 8682.941,E2 8682.941} C_VEL
LIN {X 0,Y 280.047,Z 1130.599,A -85,B 0,C 180,E1 8679.86,E2 8679.86} C_VEL
LIN {X 0,Y 290.761,Z 1114.963,A -85,B 0,C 180,E1 8677.246,E2 8677.246} C_VEL
LIN {X 0,Y 302.071,Z 1096.833,A -85,B 0,C 180,E1 8674.827,E2 8674.827} C_VEL
LIN {X 0,Y 312.088,Z 1079.048,A -85,B 0,C 180,E1 8672.925,E2 8672.925} C_VEL
LIN {X 0,Y 321.685,Z 1059.592,A -85,B 0,C 180,E1 8671.268,E2 8671.268} C_VEL
LIN {X 0,Y 330.422,Z 1039.497,A -85,B 0,C 180,E1 8669.894,E2 8669.894} C_VEL
LIN {X 0,Y 337.789,Z 1019.563,A -85,B 0,C 180,E1 8668.817,E2 8668.817} C_VEL
LIN {X 0,Y 344.91,Z 996.502,A -85,B 0,C 180,E1 8667.852,E2 8667.852} C_VEL
LIN {X 0,Y 350.333,Z 974.686,A -85,B 0,C 180,E1 8667.168,E2 8667.168} C_VEL
LIN {X 0,Y 354.419,Z 951.907,A -85,B 0,C 180,E1 8666.637,E2 8666.637} C_VEL
LIN {X 0,Y 357.274,Z 926.901,A -85,B 0,C 180,E1 8666.179,E2 8666.179} C_VEL
LIN {X 0,Y 373.027,Z 746.953,A -85,B 0,C 180,E1 8663.331,E2 8663.331} C_VEL
LIN {X 0,Y 368.832,Z 736.593,A -85,B 0,C 180,E1 8660.843,E2 8660.843} C_VEL
LIN {X 0,Y 364.847,Z 726.933,A -85,B 0,C 180,E1 8658.04,E2 8658.04} C_VEL
LIN {X 0,Y 361.242,Z 718.615,A -85,B 0,C 180,E1 8654.917,E2 8654.917} C_VEL
LIN {X 0,Y 358.479,Z 712.003,A -85,B 0,C 180,E1 8651.667,E2 8651.667} C_VEL
LIN {X 0,Y 356.761,Z 707.943,A -85,B 0,C 180,E1 8648.705,E2 8648.705} C_VEL
LIN {X 0,Y 355.826,Z 704.835,A -85,B 0,C 180,E1 8645.609,E2 8645.609} C_VEL
LIN {X 0,Y 356.038,Z 703.57,A -85,B 0,C 180,E1 8640.805,E2 8640.805} C_VEL
LIN {X 0,Y 356.261,Z 703.668,A -85,B 0,C 180,E1 8640.064,E2 8640.064} C_VEL
LIN {X 0,Y 356.633,Z 704.88,A -85,B 0,C 180,E1 8638.837,E2 8638.837} C_VEL
LIN {X 0,Y 357.148,Z 709.32,A -85,B 0,C 180,E1 8636.999,E2 8636.999} C_VEL
LIN {X 0,Y 358.048,Z 714.184,A -85,B 0,C 180,E1 8635.077,E2 8635.077} C_VEL
LIN {X 0,Y 358.353,Z 714.91,A -85,B 0,C 180,E1 8634.644,E2 8634.644} C_VEL
LIN {X 0,Y 361.088,Z 718.969,A -85,B 0,C 180,E1 8631.721,E2 8631.721} C_VEL
LIN {X 0,Y 363.966,Z 723.504,A -85,B 0,C 180,E1 8629.313,E2 8629.313} C_VEL
LIN {X 0,Y 367.838,Z 730.083,A -85,B 0,C 180,E1 8626.601,E2 8626.601} C_VEL
LIN {X 0,Y 372.121,Z 737.865,A -85,B 0,C 180,E1 8624.059,E2 8624.059} C_VEL
LIN {X 0,Y 353.234,Z 932.173,A -85,B 0,C 180,E1 8620.822,E2 8620.822} C_VEL
LIN {X 0,Y 349.323,Z 956.71,A -85,B 0,C 180,E1 8620.264,E2 8620.264} C_VEL
LIN {X 0,Y 344.742,Z 977.881,A -85,B 0,C 180,E1 8619.625,E2 8619.625} C_VEL
LIN {X 0,Y 338.493,Z 1000.473,A -85,B 0,C 180,E1 8618.739,E2 8618.739} C_VEL
LIN {X 0,Y 331.311,Z 1022.105,A -85,B 0,C 180,E1 8617.665,E2 8617.665} C_VEL
LIN {X 0,Y 322.672,Z 1043.854,A -85,B 0,C 180,E1 8616.299,E2 8616.299} C_VEL
LIN {X 0,Y 313.451,Z 1064.217,A -85,B 0,C 180,E1 8614.732,E2 8614.732} C_VEL
LIN {X 0,Y 303.346,Z 1083.649,A -85,B 0,C 180,E1 8612.866,E2 8612.866} C_VEL
LIN {X 0,Y 292.148,Z 1103.066,A -85,B 0,C 180,E1 8610.576,E2 8610.576} C_VEL
LIN {X 0,Y 281.428,Z 1119.877,A -85,B 0,C 180,E1 8608.116,E2 8608.116} C_VEL
LIN {X 0,Y 269.647,Z 1136.893,A -85,B 0,C 180,E1 8605.032,E2 8605.032} C_VEL
LIN {X 0,Y 259.255,Z 1150.913,A -85,B 0,C 180,E1 8601.883,E2 8601.883} C_VEL
LIN {X 0,Y 248.061,Z 1165.216,A -85,B 0,C 180,E1 8597.872,E2 8597.872} C_VEL
LIN {X 0,Y 238.549,Z 1176.957,A -85,B 0,C 180,E1 8593.755,E2 8593.755} C_VEL
LIN {X 0,Y 228.995,Z 1188.548,A -85,B 0,C 180,E1 8588.593,E2 8588.593} C_VEL
LIN {X 0,Y 221.314,Z 1198.172,A -85,B 0,C 180,E1 8583.138,E2 8583.138} C_VEL
LIN {X 0,Y 215.395,Z 1205.915,A -85,B 0,C 180,E1 8577.358,E2 8577.358} C_VEL
LIN {X 0,Y 211.234,Z 1212.327,A -85,B 0,C 180,E1 8571.17,E2 8571.17} C_VEL
LIN {X 0,Y 208.918,Z 1216.815,A -85,B 0,C 180,E1 8564.977,E2 8564.977} C_VEL
LIN {X 0,Y 208.088,Z 1219.603,A -85,B 0,C 180,E1 8559.402,E2 8559.402} C_VEL
LIN {X 0,Y 207.979,Z 1221.132,A -85,B 0,C 180,E1 8553.859,E2 8553.859} C_VEL
LIN {X 0,Y 208.005,Z 1221.372,A -85,B 0,C 180,E1 8548.898,E2 8548.898} C_VEL
LIN {X 0,Y 207.969,Z 1220.682,A -85,B 0,C 180,E1 8544.205,E2 8544.205} C_VEL
LIN {X 0,Y 208.2,Z 1218.973,A -85,B 0,C 180,E1 8539.205,E2 8539.205} C_VEL
LIN {X 0,Y 209.468,Z 1215.593,A -85,B 0,C 180,E1 8533.072,E2 8533.072} C_VEL
LIN {X 0,Y 212.259,Z 1210.496,A -85,B 0,C 180,E1 8526.985,E2 8526.985} C_VEL
LIN {X 0,Y 216.829,Z 1203.948,A -85,B 0,C 180,E1 8521.041,E2 8521.041} C_VEL
LIN {X 0,Y 223.235,Z 1195.558,A -85,B 0,C 180,E1 8515.332,E2 8515.332} C_VEL
LIN {X 0,Y 231.465,Z 1185.499,A -85,B 0,C 180,E1 8509.937,E2 8509.937} C_VEL
LIN {X 0,Y 240.549,Z 1174.327,A -85,B 0,C 180,E1 8505.3,E2 8505.3} C_VEL
LIN {X 0,Y 250.733,Z 1161.741,A -85,B 0,C 180,E1 8501.09,E2 8501.09} C_VEL
LIN {X 0,Y 261.617,Z 1147.563,A -85,B 0,C 180,E1 8497.35,E2 8497.35} C_VEL
LIN {X 0,Y 273.476,Z 1131.275,A -85,B 0,C 180,E1 8493.908,E2 8493.908} C_VEL
LIN {X 0,Y 283.919,Z 1115.798,A -85,B 0,C 180,E1 8491.278,E2 8491.278} C_VEL
LIN {X 0,Y 295.662,Z 1096.839,A -85,B 0,C 180,E1 8488.67,E2 8488.67} C_VEL
LIN {X 0,Y 305.552,Z 1079.214,A -85,B 0,C 180,E1 8486.704,E2 8486.704} C_VEL
LIN {X 0,Y 315.712,Z 1058.893,A -85,B 0,C 180,E1 8484.86,E2 8484.86} C_VEL
LIN {X 0,Y 324.168,Z 1039.822,A -85,B 0,C 180,E1 8483.447,E2 8483.447} C_VEL
LIN {X 0,Y 332.47,Z 1018.061,A -85,B 0,C 180,E1 8482.14,E2 8482.14} C_VEL
LIN {X 0,Y 339.268,Z 997.175,A -85,B 0,C 180,E1 8481.132,E2 8481.132} C_VEL
LIN {X 0,Y 345.439,Z 973.768,A -85,B 0,C 180,E1 8480.255,E2 8480.255} C_VEL
LIN {X 0,Y 350.218,Z 950.832,A -85,B 0,C 180,E1 8479.598,E2 8479.598} C_VEL
LIN {X 0,Y 353.587,Z 926.964,A -85,B 0,C 180,E1 8479.099,E2 8479.099} C_VEL
LIN {X 0,Y 371.857,Z 737.615,A -85,B 0,C 180,E1 8475.939,E2 8475.939} C_VEL
LIN {X 0,Y 366.792,Z 728.333,A -85,B 0,C 180,E1 8472.877,E2 8472.877} C_VEL
LIN {X 0,Y 362.538,Z 721.261,A -85,B 0,C 180,E1 8469.766,E2 8469.766} C_VEL
LIN {X 0,Y 359.845,Z 717.245,A -85,B 0,C 180,E1 8467.344,E2 8467.344} C_VEL
LIN {X 0,Y 357.51,Z 713.843,A -85,B 0,C 180,E1 8464.652,E2 8464.652} C_VEL
LIN {X 0,Y 355.213,Z 711.368,A -85,B 0,C 180,E1 8460.645,E2 8460.645} C_VEL
LIN {X 0,Y 354.4,Z 711.304,A -85,B 0,C 180,E1 8457.574,E2 8457.574} C_VEL
LIN {X 0,Y 354.659,Z 713.088,A -85,B 0,C 180,E1 8453.525,E2 8453.525} C_VEL
LIN {X 0,Y 355.935,Z 717.107,A -85,B 0,C 180,E1 8450.133,E2 8450.133} C_VEL
LIN {X 0,Y 357.883,Z 721.755,A -85,B 0,C 180,E1 8447.249,E2 8447.249} C_VEL
LIN {X 0,Y 361.083,Z 729.611,A -85,B 0,C 180,E1 8443.882,E2 8443.882} C_VEL
LIN {X 0,Y 364.009,Z 736.775,A -85,B 0,C 180,E1 8441.461,E2 8441.461} C_VEL
LIN {X 0,Y 367.681,Z 745.835,A -85,B 0,C 180,E1 8438.921,E2 8438.921} C_VEL
LIN {X 0,Y 369.701,Z 751.265,A -85,B 0,C 180,E1 8437.659,E2 8437.659} C_VEL
LIN {X 0,Y 352.33,Z 942.395,A -85,B 0,C 180,E1 8434.639,E2 8434.639} C_VEL
LIN {X 0,Y 348.605,Z 965.813,A -85,B 0,C 180,E1 8434.143,E2 8434.143} C_VEL
LIN {X 0,Y 343.693,Z 987.877,A -85,B 0,C 180,E1 8433.546,E2 8433.546} C_VEL
LIN {X 0,Y 337.711,Z 1008.513,A -85,B 0,C 180,E1 8432.791,E2 8432.791} C_VEL
LIN {X 0,Y 330.229,Z 1030.124,A -85,B 0,C 180,E1 8431.773,E2 8431.773} C_VEL
LIN {X 0,Y 322.401,Z 1049.135,A -85,B 0,C 180,E1 8430.629,E2 8430.629} C_VEL
LIN {X 0,Y 312.462,Z 1070.084,A -85,B 0,C 180,E1 8429.046,E2 8429.046} C_VEL
LIN {X 0,Y 302.809,Z 1087.991,A -85,B 0,C 180,E1 8427.351,E2 8427.351} C_VEL
LIN {X 0,Y 292.031,Z 1105.716,A -85,B 0,C 180,E1 8425.256,E2 8425.256} C_VEL
LIN {X 0,Y 281.046,Z 1122.207,A -85,B 0,C 180,E1 8422.836,E2 8422.836} C_VEL
LIN {X 0,Y 269.963,Z 1137.181,A -85,B 0,C 180,E1 8420.055,E2 8420.055} C_VEL
LIN {X 0,Y 258.418,Z 1151.725,A -85,B 0,C 180,E1 8416.669,E2 8416.669} C_VEL
LIN {X 0,Y 247.857,Z 1164.148,A -85,B 0,C 180,E1 8412.98,E2 8412.98} C_VEL
LIN {X 0,Y 237.445,Z 1175.756,A -85,B 0,C 180,E1 8408.551,E2 8408.551} C_VEL
LIN {X 0,Y 228.527,Z 1185.529,A -85,B 0,C 180,E1 8403.756,E2 8403.756} C_VEL
LIN {X 0,Y 220.89,Z 1193.735,A -85,B 0,C 180,E1 8398.378,E2 8398.378} C_VEL
LIN {X 0,Y 214.676,Z 1200.772,A -85,B 0,C 180,E1 8392.164,E2 8392.164} C_VEL
LIN {X 0,Y 210.923,Z 1205.56,A -85,B 0,C 180,E1 8386.241,E2 8386.241} C_VEL
LIN {X 0,Y 208.862,Z 1208.701,A -85,B 0,C 180,E1 8380.202,E2 8380.202} C_VEL
LIN {X 0,Y 208.152,Z 1210.349,A -85,B 0,C 180,E1 8374.684,E2 8374.684} C_VEL
LIN {X 0,Y 208.042,Z 1210.777,A -85,B 0,C 180,E1 8369.174,E2 8369.174} C_VEL
LIN {X 0,Y 208.242,Z 1210.063,A -85,B 0,C 180,E1 8363.936,E2 8363.936} C_VEL
LIN {X 0,Y 209.336,Z 1207.997,A -85,B 0,C 180,E1 8357.868,E2 8357.868} C_VEL
LIN {X 0,Y 211.871,Z 1204.285,A -85,B 0,C 180,E1 8351.852,E2 8351.852} C_VEL
LIN {X 0,Y 216.429,Z 1198.835,A -85,B 0,C 180,E1 8345.722,E2 8345.722} C_VEL
LIN {X 0,Y 222.699,Z 1191.874,A -85,B 0,C 180,E1 8340.109,E2 8340.109} C_VEL
LIN {X 0,Y 230.803,Z 1183.111,A -85,B 0,C 180,E1 8334.819,E2 8334.819} C_VEL
LIN {X 0,Y 240.156,Z 1173.006,A -85,B 0,C 180,E1 8330.122,E2 8330.122} C_VEL
LIN {X 0,Y 250.642,Z 1161.083,A -85,B 0,C 180,E1 8325.896,E2 8325.896} C_VEL
LIN {X 0,Y 262.417,Z 1147.017,A -85,B 0,C 180,E1 8322.014,E2 8322.014} C_VEL
LIN {X 0,Y 273.217,Z 1133.198,A -85,B 0,C 180,E1 8319.011,E2 8319.011} C_VEL
LIN {X 0,Y 284.558,Z 1117.322,A -85,B 0,C 180,E1 8316.275,E2 8316.275} C_VEL
LIN {X 0,Y 295.42,Z 1100.797,A -85,B 0,C 180,E1 8313.983,E2 8313.983} C_VEL
LIN {X 0,Y 305.948,Z 1082.749,A -85,B 0,C 180,E1 8311.999,E2 8311.999} C_VEL
LIN {X 0,Y 316.463,Z 1062.498,A -85,B 0,C 180,E1 8310.218,E2 8310.218} C_VEL
LIN {X 0,Y 324.953,Z 1043.81,A -85,B 0,C 180,E1 8308.91,E2 8308.91} C_VEL
LIN {X 0,Y 333.225,Z 1022.545,A -85,B 0,C 180,E1 8307.729,E2 8307.729} C_VEL
LIN {X 0,Y 340.235,Z 1001.292,A -85,B 0,C 180,E1 8306.806,E2 8306.806} C_VEL
LIN {X 0,Y 346.05,Z 978.995,A -85,B 0,C 180,E1 8306.086,E2 8306.086} C_VEL
LIN {X 0,Y 350.806,Z 954.85,A -85,B 0,C 180,E1 8305.502,E2 8305.502} C_VEL
LIN {X 0,Y 353.682,Z 932.343,A -85,B 0,C 180,E1 8305.077,E2 8305.077} C_VEL
LIN {X 0,Y 369.953,Z 751.295,A -85,B 0,C 180,E1 8302.234,E2 8302.234} C_VEL
LIN {X 0,Y 365.718,Z 740.45,A -85,B 0,C 180,E1 8299.485,E2 8299.485} C_VEL
LIN {X 0,Y 362.013,Z 731.444,A -85,B 0,C 180,E1 8296.611,E2 8296.611} C_VEL
LIN {X 0,Y 359.409,Z 725.173,A -85,B 0,C 180,E1 8294.089,E2 8294.089} C_VEL
LIN {X 0,Y 357.224,Z 719.604,A -85,B 0,C 180,E1 8291.299,E2 8291.299} C_VEL
LIN {X 0,Y 355.644,Z 715.673,A -85,B 0,C 180,E1 8288.407,E2 8288.407} C_VEL
LIN {X 0,Y 354.827,Z 712.744,A -85,B 0,C 180,E1 8285.498,E2 8285.498} C_VEL
LIN {X 0,Y 355.063,Z 711.512,A -85,B 0,C 180,E1 8280.807,E2 8280.807} C_VEL
LIN {X 0,Y 356.189,Z 712.418,A -85,B 0,C 180,E1 8277.909,E2 8277.909} C_VEL
LIN {X 0,Y 358.24,Z 714.691,A -85,B 0,C 180,E1 8274.795,E2 8274.795} C_VEL
LIN {X 0,Y 358.353,Z 714.91,A -85,B 0,C 180,E1 8274.644,E2 8274.644} C_VEL
LIN {X 0,Y 359.187,Z 717.564,A -85,B 0,C 180,E1 8273.486,E2 8273.486} C_VEL
LIN {X 0,Y 361.733,Z 729.44,A -85,B 0,C 180,E1 8270.278,E2 8270.278} C_VEL
LIN {X 0,Y 362.49,Z 731.109,A -85,B 0,C 180,E1 8269.631,E2 8269.631} C_VEL
LIN {X 0,Y 366.44,Z 738.042,A -85,B 0,C 180,E1 8266.79,E2 8266.79} C_VEL
LIN {X 0,Y 369.04,Z 743.182,A -85,B 0,C 180,E1 8265.147,E2 8265.147} C_VEL
LIN {X 0,Y 350.263,Z 932.551,A -85,B 0,C 180,E1 8262.03,E2 8262.03} C_VEL
LIN {X 0,Y 346.31,Z 956.898,A -85,B 0,C 180,E1 8261.486,E2 8261.486} C_VEL
LIN {X 0,Y 341.668,Z 977.985,A -85,B 0,C 180,E1 8260.863,E2 8260.863} C_VEL
LIN {X 0,Y 335.209,Z 1000.898,A -85,B 0,C 180,E1 8259.98,E2 8259.98} C_VEL
LIN {X 0,Y 327.89,Z 1022.5,A -85,B 0,C 180,E1 8258.924,E2 8258.924} C_VEL
LIN {X 0,Y 319.501,Z 1043.214,A -85,B 0,C 180,E1 8257.647,E2 8257.647} C_VEL
LIN {X 0,Y 310.041,Z 1063.75,A -85,B 0,C 180,E1 8256.101,E2 8256.101} C_VEL
LIN {X 0,Y 299.689,Z 1083.231,A -85,B 0,C 180,E1 8254.264,E2 8254.264} C_VEL
LIN {X 0,Y 288.558,Z 1102.151,A -85,B 0,C 180,E1 8252.077,E2 8252.077} C_VEL
LIN {X 0,Y 277.505,Z 1119.033,A -85,B 0,C 180,E1 8249.646,E2 8249.646} C_VEL
LIN {X 0,Y 264.99,Z 1136.608,A -85,B 0,C 180,E1 8246.499,E2 8246.499} C_VEL
LIN {X 0,Y 254.221,Z 1150.642,A -85,B 0,C 180,E1 8243.354,E2 8243.354} C_VEL
LIN {X 0,Y 242.565,Z 1164.964,A -85,B 0,C 180,E1 8239.328,E2 8239.328} C_VEL
LIN {X 0,Y 232.62,Z 1176.713,A -85,B 0,C 180,E1 8235.171,E2 8235.171} C_VEL
LIN {X 0,Y 222.619,Z 1188.257,A -85,B 0,C 180,E1 8229.96,E2 8229.96} C_VEL
LIN {X 0,Y 214.421,Z 1197.947,A -85,B 0,C 180,E1 8224.349,E2 8224.349} C_VEL
LIN {X 0,Y 208.095,Z 1205.699,A -85,B 0,C 180,E1 8218.403,E2 8218.403} C_VEL
LIN {X 0,Y 203.703,Z 1211.935,A -85,B 0,C 180,E1 8212.206,E2 8212.206} C_VEL
LIN {X 0,Y 201.128,Z 1216.437,A -85,B 0,C 180,E1 8205.868,E2 8205.868} C_VEL
LIN {X 0,Y 200.133,Z 1219.275,A -85,B 0,C 180,E1 8200.07,E2 8200.07} C_VEL
LIN {X 0,Y 199.975,Z 1220.902,A -85,B 0,C 180,E1 8194.301,E2 8194.301} C_VEL
LIN {X 0,Y 200.009,Z 1221.181,A -85,B 0,C 180,E1 8189.015,E2 8189.015} C_VEL
LIN {X 0,Y 199.976,Z 1220.476,A -85,B 0,C 180,E1 8183.973,E2 8183.973} C_VEL
LIN {X 0,Y 200.24,Z 1218.765,A -85,B 0,C 180,E1 8178.771,E2 8178.771} C_VEL
LIN {X 0,Y 201.657,Z 1215.382,A -85,B 0,C 180,E1 8172.395,E2 8172.395} C_VEL
LIN {X 0,Y 204.819,Z 1210.119,A -85,B 0,C 180,E1 8165.91,E2 8165.91} C_VEL
LIN {X 0,Y 209.891,Z 1203.397,A -85,B 0,C 180,E1 8159.672,E2 8159.672} C_VEL
LIN {X 0,Y 216.849,Z 1194.868,A -85,B 0,C 180,E1 8153.797,E2 8153.797} C_VEL
LIN {X 0,Y 225.61,Z 1184.728,A -85,B 0,C 180,E1 8148.336,E2 8148.336} C_VEL
LIN {X 0,Y 235.106,Z 1173.626,A -85,B 0,C 180,E1 8143.699,E2 8143.699} C_VEL
LIN {X 0,Y 246.497,Z 1160.036,A -85,B 0,C 180,E1 8139.218,E2 8139.218} C_VEL
LIN {X 0,Y 257.3,Z 1146.495,A -85,B 0,C 180,E1 8135.692,E2 8135.692} C_VEL
LIN {X 0,Y 269.618,Z 1130.016,A -85,B 0,C 180,E1 8132.273,E2 8132.273} C_VEL
LIN {X 0,Y 280.652,Z 1114.113,A -85,B 0,C 180,E1 8129.625,E2 8129.625} C_VEL
LIN {X 0,Y 292.205,Z 1095.769,A -85,B 0,C 180,E1 8127.17,E2 8127.17} C_VEL
LIN {X 0,Y 302.715,Z 1077.432,A -85,B 0,C 180,E1 8125.175,E2 8125.175} C_VEL
LIN {X 0,Y 312.746,Z 1057.549,A -85,B 0,C 180,E1 8123.43,E2 8123.43} C_VEL
LIN {X 0,Y 321.849,Z 1037.304,A -85,B 0,C 180,E1 8121.979,E2 8121.979} C_VEL
LIN {X 0,Y 330.057,Z 1015.675,A -85,B 0,C 180,E1 8120.741,E2 8120.741} C_VEL
LIN {X 0,Y 337.436,Z 992.719,A -85,B 0,C 180,E1 8119.691,E2 8119.691} C_VEL
LIN {X 0,Y 343.111,Z 970.746,A -85,B 0,C 180,E1 8118.918,E2 8118.918} C_VEL
LIN {X 0,Y 348.083,Z 945.505,A -85,B 0,C 180,E1 8118.251,E2 8118.251} C_VEL
LIN {X 0,Y 351.23,Z 922.133,A -85,B 0,C 180,E1 8117.798,E2 8117.798} C_VEL
LIN {X 0,Y 368.789,Z 742.698,A -85,B 0,C 180,E1 8114.846,E2 8114.846} C_VEL
LIN {X 0,Y 364.672,Z 735.029,A -85,B 0,C 180,E1 8112.188,E2 8112.188} C_VEL
LIN {X 0,Y 360.862,Z 728.546,A -85,B 0,C 180,E1 8109.248,E2 8109.248} C_VEL
LIN {X 0,Y 358.45,Z 724.833,A -85,B 0,C 180,E1 8106.97,E2 8106.97} C_VEL
LIN {X 0,Y 356.396,Z 721.715,A -85,B 0,C 180,E1 8104.506,E2 8104.506} C_VEL
LIN {X 0,Y 354.174,Z 719.266,A -85,B 0,C 180,E1 8100.485,E2 8100.485} C_VEL
LIN {X 0,Y 353.405,Z 719.298,A -85,B 0,C 180,E1 8097.405,E2 8097.405} C_VEL
LIN {X 0,Y 353.641,Z 720.995,A -85,B 0,C 180,E1 8093.669,E2 8093.669} C_VEL
LIN {X 0,Y 354.82,Z 724.934,A -85,B 0,C 180,E1 8090.347,E2 8090.347} C_VEL
LIN {X 0,Y 356.586,Z 729.319,A -85,B 0,C 180,E1 8087.613,E2 8087.613} C_VEL
LIN {X 0,Y 359.567,Z 736.996,A -85,B 0,C 180,E1 8084.31,E2 8084.31} C_VEL
LIN {X 0,Y 362.338,Z 744.077,A -85,B 0,C 180,E1 8081.914,E2 8081.914} C_VEL
LIN {X 0,Y 365.698,Z 752.755,A -85,B 0,C 180,E1 8079.472,E2 8079.472} C_VEL
LIN {X 0,Y 366.725,Z 755.877,A -85,B 0,C 180,E1 8078.772,E2 8078.772} C_VEL
LIN {X 0,Y 349.372,Z 942.193,A -85,B 0,C 180,E1 8075.857,E2 8075.857} C_VEL
LIN {X 0,Y 345.57,Z 965.628,A -85,B 0,C 180,E1 8075.369,E2 8075.369} C_VEL
LIN {X 0,Y 340.434,Z 988.18,A -85,B 0,C 180,E1 8074.769,E2 8074.769} C_VEL
LIN {X 0,Y 334.339,Z 1008.79,A -85,B 0,C 180,E1 8074.029,E2 8074.029} C_VEL
LIN {X 0,Y 326.534,Z 1030.772,A -85,B 0,C 180,E1 8073.006,E2 8073.006} C_VEL
LIN {X 0,Y 318.561,Z 1049.704,A -85,B 0,C 180,E1 8071.88,E2 8071.88} C_VEL
LIN {X 0,Y 308.421,Z 1070.537,A -85,B 0,C 180,E1 8070.321,E2 8070.321} C_VEL
LIN {X 0,Y 298.188,Z 1089.061,A -85,B 0,C 180,E1 8068.58,E2 8068.58} C_VEL
LIN {X 0,Y 287.166,Z 1106.607,A -85,B 0,C 180,E1 8066.501,E2 8066.501} C_VEL
LIN {X 0,Y 276.254,Z 1122.505,A -85,B 0,C 180,E1 8064.167,E2 8064.167} C_VEL
LIN {X 0,Y 264.853,Z 1137.46,A -85,B 0,C 180,E1 8061.394,E2 8061.394} C_VEL
LIN {X 0,Y 252.936,Z 1151.976,A -85,B 0,C 180,E1 8058.002,E2 8058.002} C_VEL
LIN {X 0,Y 242.541,Z 1163.767,A -85,B 0,C 180,E1 8054.492,E2 8054.492} C_VEL
LIN {X 0,Y 231.64,Z 1175.483,A -85,B 0,C 180,E1 8050.027,E2 8050.027} C_VEL
LIN {X 0,Y 222.233,Z 1185.325,A -85,B 0,C 180,E1 8045.162,E2 8045.162} C_VEL
LIN {X 0,Y 214.107,Z 1193.61,A -85,B 0,C 180,E1 8039.67,E2 8039.67} C_VEL
LIN {X 0,Y 207.652,Z 1200.492,A -85,B 0,C 180,E1 8033.556,E2 8033.556} C_VEL
LIN {X 0,Y 203.566,Z 1205.225,A -85,B 0,C 180,E1 8027.653,E2 8027.653} C_VEL
LIN {X 0,Y 201.012,Z 1208.798,A -85,B 0,C 180,E1 8020.895,E2 8020.895} C_VEL
LIN {X 0,Y 200.184,Z 1210.489,A -85,B 0,C 180,E1 8015.158,E2 8015.158} C_VEL
LIN {X 0,Y 200.043,Z 1211.003,A -85,B 0,C 180,E1 8009.427,E2 8009.427} C_VEL
LIN {X 0,Y 200.239,Z 1210.333,A -85,B 0,C 180,E1 8003.981,E2 8003.981} C_VEL
LIN {X 0,Y 201.29,Z 1208.429,A -85,B 0,C 180,E1 7997.958,E2 7997.958} C_VEL
LIN {X 0,Y 204.03,Z 1204.691,A -85,B 0,C 180,E1 7991.426,E2 7991.426} C_VEL
LIN {X 0,Y 208.805,Z 1199.34,A -85,B 0,C 180,E1 7985.078,E2 7985.078} C_VEL
LIN {X 0,Y 215.352,Z 1192.429,A -85,B 0,C 180,E1 7979.288,E2 7979.288} C_VEL
LIN {X 0,Y 224.214,Z 1183.329,A -85,B 0,C 180,E1 7973.623,E2 7973.623} C_VEL
LIN {X 0,Y 233.988,Z 1173.232,A -85,B 0,C 180,E1 7968.848,E2 7968.848} C_VEL
LIN {X 0,Y 244.629,Z 1161.612,A -85,B 0,C 180,E1 7964.669,E2 7964.669} C_VEL
LIN {X 0,Y 256.457,Z 1148.035,A -85,B 0,C 180,E1 7960.856,E2 7960.856} C_VEL
LIN {X 0,Y 267.33,Z 1134.574,A -85,B 0,C 180,E1 7957.892,E2 7957.892} C_VEL
LIN {X 0,Y 279.562,Z 1118.073,A -85,B 0,C 180,E1 7955.013,E2 7955.013} C_VEL
LIN {X 0,Y 291.005,Z 1101.148,A -85,B 0,C 180,E1 7952.671,E2 7952.671} C_VEL
LIN {X 0,Y 301.776,Z 1083.148,A -85,B 0,C 180,E1 7950.708,E2 7950.708} C_VEL
LIN {X 0,Y 312.127,Z 1063.796,A -85,B 0,C 180,E1 7949.012,E2 7949.012} C_VEL
LIN {X 0,Y 321.169,Z 1044.367,A -85,B 0,C 180,E1 7947.663,E2 7947.663} C_VEL
LIN {X 0,Y 329.593,Z 1023.276,A -85,B 0,C 180,E1 7946.503,E2 7946.503} C_VEL
LIN {X 0,Y 336.542,Z 1002.718,A -85,B 0,C 180,E1 7945.619,E2 7945.619} C_VEL
LIN {X 0,Y 342.579,Z 980.449,A -85,B 0,C 180,E1 7944.899,E2 7944.899} C_VEL
LIN {X 0,Y 347.336,Z 957.752,A -85,B 0,C 180,E1 7944.344,E2 7944.344} C_VEL
LIN {X 0,Y 350.414,Z 935.189,A -85,B 0,C 180,E1 7943.914,E2 7943.914} C_VEL
LIN {X 0,Y 366.99,Z 755.805,A -85,B 0,C 180,E1 7941.116,E2 7941.116} C_VEL
LIN {X 0,Y 363.207,Z 745.855,A -85,B 0,C 180,E1 7938.457,E2 7938.457} C_VEL
LIN {X 0,Y 360.302,Z 738.417,A -85,B 0,C 180,E1 7936.029,E2 7936.029} C_VEL
LIN {X 0,Y 357.992,Z 732.569,A -85,B 0,C 180,E1 7933.651,E2 7933.651} C_VEL
LIN {X 0,Y 355.984,Z 727.203,A -85,B 0,C 180,E1 7930.929,E2 7930.929} C_VEL
LIN {X 0,Y 354.562,Z 723.482,A -85,B 0,C 180,E1 7928.186,E2 7928.186} C_VEL
LIN {X 0,Y 353.824,Z 720.638,A -85,B 0,C 180,E1 7925.351,E2 7925.351} C_VEL
LIN {X 0,Y 354.088,Z 719.454,A -85,B 0,C 180,E1 7920.809,E2 7920.809} C_VEL
LIN {X 0,Y 355.196,Z 720.394,A -85,B 0,C 180,E1 7917.903,E2 7917.903} C_VEL
LIN {X 0,Y 357.139,Z 722.647,A -85,B 0,C 180,E1 7914.906,E2 7914.906} C_VEL
LIN {X 0,Y 359.828,Z 726.786,A -85,B 0,C 180,E1 7911.933,E2 7911.933} C_VEL
LIN {X 0,Y 362.49,Z 731.109,A -85,B 0,C 180,E1 7909.631,E2 7909.631} C_VEL
LIN {X 0,Y 363.27,Z 733.673,A -85,B 0,C 180,E1 7908.929,E2 7908.929} C_VEL
LIN {X 0,Y 364.715,Z 744.531,A -85,B 0,C 180,E1 7907.265,E2 7907.265} C_VEL
LIN {X 0,Y 365.357,Z 746.561,A -85,B 0,C 180,E1 7906.775,E2 7906.775} C_VEL
LIN {X 0,Y 366.117,Z 748.346,A -85,B 0,C 180,E1 7906.256,E2 7906.256} C_VEL
LIN {X 0,Y 347.452,Z 932.901,A -85,B 0,C 180,E1 7903.259,E2 7903.259} C_VEL
LIN {X 0,Y 343.41,Z 957.329,A -85,B 0,C 180,E1 7902.723,E2 7902.723} C_VEL
LIN {X 0,Y 338.586,Z 978.807,A -85,B 0,C 180,E1 7902.098,E2 7902.098} C_VEL
LIN {X 0,Y 332.087,Z 1001.324,A -85,B 0,C 180,E1 7901.245,E2 7901.245} C_VEL
LIN {X 0,Y 324.461,Z 1023.363,A -85,B 0,C 180,E1 7900.185,E2 7900.185} C_VEL
LIN {X 0,Y 315.638,Z 1044.535,A -85,B 0,C 180,E1 7898.891,E2 7898.891} C_VEL
LIN {X 0,Y 306.015,Z 1064.796,A -85,B 0,C 180,E1 7897.372,E2 7897.372} C_VEL
LIN {X 0,Y 295.44,Z 1084.175,A -85,B 0,C 180,E1 7895.557,E2 7895.557} C_VEL
LIN {X 0,Y 283.296,Z 1104.062,A -85,B 0,C 180,E1 7893.244,E2 7893.244} C_VEL
LIN {X 0,Y 271.996,Z 1120.773,A -85,B 0,C 180,E1 7890.815,E2 7890.815} C_VEL
LIN {X 0,Y 259.837,Z 1137.187,A -85,B 0,C 180,E1 7887.84,E2 7887.84} C_VEL
LIN {X 0,Y 248.101,Z 1151.944,A -85,B 0,C 180,E1 7884.495,E2 7884.495} C_VEL
LIN {X 0,Y 236.089,Z 1166.021,A -85,B 0,C 180,E1 7880.424,E2 7880.424} C_VEL
LIN {X 0,Y 225.309,Z 1178.235,A -85,B 0,C 180,E1 7875.964,E2 7875.964} C_VEL
LIN {X 0,Y 215.362,Z 1189.071,A -85,B 0,C 180,E1 7870.818,E2 7870.818} C_VEL
LIN {X 0,Y 206.931,Z 1198.496,A -85,B 0,C 180,E1 7865.099,E2 7865.099} C_VEL
LIN {X 0,Y 200.35,Z 1206.115,A -85,B 0,C 180,E1 7858.952,E2 7858.952} C_VEL
LIN {X 0,Y 195.62,Z 1212.407,A -85,B 0,C 180,E1 7852.224,E2 7852.224} C_VEL
LIN {X 0,Y 193.119,Z 1216.564,A -85,B 0,C 180,E1 7845.926,E2 7845.926} C_VEL
LIN {X 0,Y 192.079,Z 1219.545,A -85,B 0,C 180,E1 7839.286,E2 7839.286} C_VEL
LIN {X 0,Y 191.983,Z 1220.798,A -85,B 0,C 180,E1 7833.284,E2 7833.284} C_VEL
LIN {X 0,Y 192.007,Z 1220.939,A -85,B 0,C 180,E1 7828.508,E2 7828.508} C_VEL
LIN {X 0,Y 191.992,Z 1220.198,A -85,B 0,C 180,E1 7823.421,E2 7823.421} C_VEL
LIN {X 0,Y 192.331,Z 1218.437,A -85,B 0,C 180,E1 7817.998,E2 7817.998} C_VEL
LIN {X 0,Y 194.1,Z 1214.744,A -85,B 0,C 180,E1 7811.063,E2 7811.063} C_VEL
LIN {X 0,Y 197.403,Z 1209.799,A -85,B 0,C 180,E1 7804.82,E2 7804.82} C_VEL
LIN {X 0,Y 202.789,Z 1203.175,A -85,B 0,C 180,E1 7798.491,E2 7798.491} C_VEL
LIN {X 0,Y 210.169,Z 1194.684,A -85,B 0,C 180,E1 7792.487,E2 7792.487} C_VEL
LIN {X 0,Y 219.474,Z 1184.488,A -85,B 0,C 180,E1 7786.894,E2 7786.894} C_VEL
LIN {X 0,Y 229.671,Z 1173.127,A -85,B 0,C 180,E1 7782.102,E2 7782.102} C_VEL
LIN {X 0,Y 241.937,Z 1159.052,A -85,B 0,C 180,E1 7777.488,E2 7777.488} C_VEL
LIN {X 0,Y 253.206,Z 1145.433,A -85,B 0,C 180,E1 7773.979,E2 7773.979} C_VEL
LIN {X 0,Y 265.641,Z 1129.232,A -85,B 0,C 180,E1 7770.677,E2 7770.677} C_VEL
LIN {X 0,Y 277.395,Z 1112.75,A -85,B 0,C 180,E1 7767.983,E2 7767.983} C_VEL
LIN {X 0,Y 289.002,Z 1094.62,A -85,B 0,C 180,E1 7765.625,E2 7765.625} C_VEL
LIN {X 0,Y 300.089,Z 1075.57,A -85,B 0,C 180,E1 7763.614,E2 7763.614} C_VEL
LIN {X 0,Y 309.987,Z 1056.188,A -85,B 0,C 180,E1 7761.973,E2 7761.973} C_VEL
LIN {X 0,Y 319.54,Z 1034.997,A -85,B 0,C 180,E1 7760.516,E2 7760.516} C_VEL
LIN {X 0,Y 327.08,Z 1015.394,A -85,B 0,C 180,E1 7759.428,E2 7759.428} C_VEL
LIN {X 0,Y 334.446,Z 992.847,A -85,B 0,C 180,E1 7758.421,E2 7758.421} C_VEL
LIN {X 0,Y 340.239,Z 970.781,A -85,B 0,C 180,E1 7757.661,E2 7757.661} C_VEL
LIN {X 0,Y 345.263,Z 945.631,A -85,B 0,C 180,E1 7757.013,E2 7757.013} C_VEL
LIN {X 0,Y 348.464,Z 922.227,A -85,B 0,C 180,E1 7756.567,E2 7756.567} C_VEL
LIN {X 0,Y 365.827,Z 747.791,A -85,B 0,C 180,E1 7753.716,E2 7753.716} C_VEL
LIN {X 0,Y 361.742,Z 740.085,A -85,B 0,C 180,E1 7750.834,E2 7750.834} C_VEL
LIN {X 0,Y 358.79,Z 735.144,A -85,B 0,C 180,E1 7748.332,E2 7748.332} C_VEL
LIN {X 0,Y 356.998,Z 732.315,A -85,B 0,C 180,E1 7746.513,E2 7746.513} C_VEL
LIN {X 0,Y 355.285,Z 729.588,A -85,B 0,C 180,E1 7744.358,E2 7744.358} C_VEL
LIN {X 0,Y 353.198,Z 727.214,A -85,B 0,C 180,E1 7740.487,E2 7740.487} C_VEL
LIN {X 0,Y 352.45,Z 727.205,A -85,B 0,C 180,E1 7737.561,E2 7737.561} C_VEL
LIN {X 0,Y 352.601,Z 728.708,A -85,B 0,C 180,E1 7733.977,E2 7733.977} C_VEL
LIN {X 0,Y 353.714,Z 732.761,A -85,B 0,C 180,E1 7730.563,E2 7730.563} C_VEL
LIN {X 0,Y 355.358,Z 737.064,A -85,B 0,C 180,E1 7727.9,E2 7727.9} C_VEL
LIN {X 0,Y 358.111,Z 744.487,A -85,B 0,C 180,E1 7724.701,E2 7724.701} C_VEL
LIN {X 0,Y 360.682,Z 751.378,A -85,B 0,C 180,E1 7722.37,E2 7722.37} C_VEL
LIN {X 0,Y 363.804,Z 759.836,A -85,B 0,C 180,E1 7719.99,E2 7719.99} C_VEL
LIN {X 0,Y 363.873,Z 760.641,A -85,B 0,C 180,E1 7719.901,E2 7719.901} C_VEL
LIN {X 0,Y 346.572,Z 941.988,A -85,B 0,C 180,E1 7717.096,E2 7717.096} C_VEL
LIN {X 0,Y 342.684,Z 965.496,A -85,B 0,C 180,E1 7716.615,E2 7716.615} C_VEL
LIN {X 0,Y 337.546,Z 987.741,A -85,B 0,C 180,E1 7716.038,E2 7716.038} C_VEL
LIN {X 0,Y 331.249,Z 1008.686,A -85,B 0,C 180,E1 7715.306,E2 7715.306} C_VEL
LIN {X 0,Y 323.402,Z 1030.419,A -85,B 0,C 180,E1 7714.319,E2 7714.319} C_VEL
LIN {X 0,Y 315.317,Z 1049.288,A -85,B 0,C 180,E1 7713.225,E2 7713.225} C_VEL
LIN {X 0,Y 304.929,Z 1070.26,A -85,B 0,C 180,E1 7711.691,E2 7711.691} C_VEL
LIN {X 0,Y 294.848,Z 1088.15,A -85,B 0,C 180,E1 7710.045,E2 7710.045} C_VEL
LIN {X 0,Y 283.549,Z 1105.856,A -85,B 0,C 180,E1 7708.001,E2 7708.001} C_VEL
LIN {X 0,Y 272.326,Z 1121.866,A -85,B 0,C 180,E1 7705.7,E2 7705.7} C_VEL
LIN {X 0,Y 260.558,Z 1136.919,A -85,B 0,C 180,E1 7702.952,E2 7702.952} C_VEL
LIN {X 0,Y 248.852,Z 1150.852,A -85,B 0,C 180,E1 7699.764,E2 7699.764} C_VEL
LIN {X 0,Y 237.401,Z 1163.389,A -85,B 0,C 180,E1 7696.071,E2 7696.071} C_VEL
LIN {X 0,Y 225.489,Z 1175.709,A -85,B 0,C 180,E1 7691.353,E2 7691.353} C_VEL
LIN {X 0,Y 215.647,Z 1185.55,A -85,B 0,C 180,E1 7686.404,E2 7686.404} C_VEL
LIN {X 0,Y 207.091,Z 1193.826,A -85,B 0,C 180,E1 7680.782,E2 7680.782} C_VEL
LIN {X 0,Y 200.243,Z 1200.703,A -85,B 0,C 180,E1 7674.484,E2 7674.484} C_VEL
LIN {X 0,Y 195.779,Z 1205.549,A -85,B 0,C 180,E1 7668.204,E2 7668.204} C_VEL
LIN {X 0,Y 193.111,Z 1209.004,A -85,B 0,C 180,E1 7661.347,E2 7661.347} C_VEL
LIN {X 0,Y 192.2,Z 1210.694,A -85,B 0,C 180,E1 7655.373,E2 7655.373} C_VEL
LIN {X 0,Y 192.045,Z 1211.208,A -85,B 0,C 180,E1 7649.403,E2 7649.403} C_VEL
LIN {X 0,Y 192.262,Z 1210.537,A -85,B 0,C 180,E1 7643.73,E2 7643.73} C_VEL
LIN {X 0,Y 193.413,Z 1208.634,A -85,B 0,C 180,E1 7637.46,E2 7637.46} C_VEL
LIN {X 0,Y 196.372,Z 1204.898,A -85,B 0,C 180,E1 7630.673,E2 7630.673} C_VEL
LIN {X 0,Y 201.475,Z 1199.552,A -85,B 0,C 180,E1 7624.106,E2 7624.106} C_VEL
LIN {X 0,Y 208.494,Z 1192.563,A -85,B 0,C 180,E1 7618.088,E2 7618.088} C_VEL
LIN {X 0,Y 217.729,Z 1183.551,A -85,B 0,C 180,E1 7612.355,E2 7612.355} C_VEL
LIN {X 0,Y 228.168,Z 1173.233,A -85,B 0,C 180,E1 7607.411,E2 7607.411} C_VEL
LIN {X 0,Y 239.003,Z 1161.851,A -85,B 0,C 180,E1 7603.288,E2 7603.288} C_VEL
LIN {X 0,Y 250.608,Z 1149.053,A -85,B 0,C 180,E1 7599.645,E2 7599.645} C_VEL
LIN {X 0,Y 261.772,Z 1135.678,A -85,B 0,C 180,E1 7596.668,E2 7596.668} C_VEL
LIN {X 0,Y 274.306,Z 1119.383,A -85,B 0,C 180,E1 7593.791,E2 7593.791} C_VEL
LIN {X 0,Y 285.253,Z 1103.678,A -85,B 0,C 180,E1 7591.597,E2 7591.597} C_VEL
LIN {X 0,Y 296.608,Z 1085.527,A -85,B 0,C 180,E1 7589.575,E2 7589.575} C_VEL
LIN {X 0,Y 307.142,Z 1066.64,A -85,B 0,C 180,E1 7587.893,E2 7587.893} C_VEL
LIN {X 0,Y 316.733,Z 1046.708,A -85,B 0,C 180,E1 7586.498,E2 7586.498} C_VEL
LIN {X 0,Y 325.297,Z 1026.252,A -85,B 0,C 180,E1 7585.357,E2 7585.357} C_VEL
LIN {X 0,Y 332.342,Z 1006.129,A -85,B 0,C 180,E1 7584.484,E2 7584.484} C_VEL
LIN {X 0,Y 339.023,Z 982.876,A -85,B 0,C 180,E1 7583.716,E2 7583.716} C_VEL
LIN {X 0,Y 343.833,Z 961.126,A -85,B 0,C 180,E1 7583.179,E2 7583.179} C_VEL
LIN {X 0,Y 347.323,Z 937.754,A -85,B 0,C 180,E1 7582.725,E2 7582.725} C_VEL
LIN {X 0,Y 364.14,Z 760.258,A -85,B 0,C 180,E1 7579.961,E2 7579.961} C_VEL
LIN {X 0,Y 360.907,Z 751.488,A -85,B 0,C 180,E1 7577.494,E2 7577.494} C_VEL
LIN {X 0,Y 358.348,Z 744.64,A -85,B 0,C 180,E1 7575.16,E2 7575.16} C_VEL
LIN {X 0,Y 356.034,Z 738.433,A -85,B 0,C 180,E1 7572.489,E2 7572.489} C_VEL
LIN {X 0,Y 354.552,Z 734.354,A -85,B 0,C 180,E1 7570.234,E2 7570.234} C_VEL
LIN {X 0,Y 353.486,Z 731.294,A -85,B 0,C 180,E1 7567.967,E2 7567.967} C_VEL
LIN {X 0,Y 352.823,Z 728.534,A -85,B 0,C 180,E1 7565.203,E2 7565.203} C_VEL
LIN {X 0,Y 353.154,Z 727.406,A -85,B 0,C 180,E1 7560.649,E2 7560.649} C_VEL
LIN {X 0,Y 354.204,Z 728.37,A -85,B 0,C 180,E1 7557.897,E2 7557.897} C_VEL
LIN {X 0,Y 355.934,Z 730.389,A -85,B 0,C 180,E1 7555.166,E2 7555.166} C_VEL
LIN {X 0,Y 358.573,Z 734.602,A -85,B 0,C 180,E1 7552.147,E2 7552.147} C_VEL
LIN {X 0,Y 361.216,Z 739.038,A -85,B 0,C 180,E1 7549.796,E2 7549.796} C_VEL
LIN {X 0,Y 365.048,Z 745.989,A -85,B 0,C 180,E1 7546.98,E2 7546.98} C_VEL
LIN {X 0,Y 365.357,Z 746.561,A -85,B 0,C 180,E1 7546.775,E2 7546.775} C_VEL
LIN {X 0,Y 365.589,Z 748.421,A -85,B 0,C 180,E1 7546.524,E2 7546.524} C_VEL
LIN {X 0,Y 365.329,Z 751.706,A -85,B 0,C 180,E1 7546.435,E2 7546.435} C_VEL
LIN {X 0,Y 364.402,Z 756.668,A -85,B 0,C 180,E1 7546.577,E2 7546.577} C_VEL
LIN {X 0,Y 362.27,Z 765.817,A -85,B 0,C 180,E1 7547.074,E2 7547.074} C_VEL
LIN {X 0,Y 361.606,Z 770.162,A -85,B 0,C 180,E1 7547.124,E2 7547.124} C_VEL
LIN {X 0,Y 344.807,Z 933.222,A -85,B 0,C 180,E1 7544.508,E2 7544.508} C_VEL
LIN {X 0,Y 340.706,Z 957.593,A -85,B 0,C 180,E1 7543.984,E2 7543.984} C_VEL
LIN {X 0,Y 335.803,Z 979.055,A -85,B 0,C 180,E1 7543.375,E2 7543.375} C_VEL
LIN {X 0,Y 329.129,Z 1001.751,A -85,B 0,C 180,E1 7542.534,E2 7542.534} C_VEL
LIN {X 0,Y 321.367,Z 1023.74,A -85,B 0,C 180,E1 7541.497,E2 7541.497} C_VEL
LIN {X 0,Y 312.372,Z 1044.875,A -85,B 0,C 180,E1 7540.229,E2 7540.229} C_VEL
LIN {X 0,Y 302.55,Z 1065.087,A -85,B 0,C 180,E1 7538.739,E2 7538.739} C_VEL
LIN {X 0,Y 292.139,Z 1083.762,A -85,B 0,C 180,E1 7537.023,E2 7537.023} C_VEL
LIN {X 0,Y 280.071,Z 1103.151,A -85,B 0,C 180,E1 7534.823,E2 7534.823} C_VEL
LIN {X 0,Y 268.961,Z 1119.196,A -85,B 0,C 180,E1 7532.549,E2 7532.549} C_VEL
LIN {X 0,Y 255.53,Z 1136.898,A -85,B 0,C 180,E1 7529.41,E2 7529.41} C_VEL
LIN {X 0,Y 244.035,Z 1150.882,A -85,B 0,C 180,E1 7526.277,E2 7526.277} C_VEL
LIN {X 0,Y 231.481,Z 1165.121,A -85,B 0,C 180,E1 7522.227,E2 7522.227} C_VEL
LIN {X 0,Y 220.147,Z 1177.408,A -85,B 0,C 180,E1 7517.758,E2 7517.758} C_VEL
LIN {X 0,Y 209.698,Z 1188.272,A -85,B 0,C 180,E1 7512.615,E2 7512.615} C_VEL
LIN {X 0,Y 200.575,Z 1197.906,A -85,B 0,C 180,E1 7506.741,E2 7506.741} C_VEL
LIN {X 0,Y 193.438,Z 1205.582,A -85,B 0,C 180,E1 7500.434,E2 7500.434} C_VEL
LIN {X 0,Y 188.21,Z 1211.979,A -85,B 0,C 180,E1 7493.48,E2 7493.48} C_VEL
LIN {X 0,Y 185.284,Z 1216.356,A -85,B 0,C 180,E1 7486.619,E2 7486.619} C_VEL
LIN {X 0,Y 184.102,Z 1219.338,A -85,B 0,C 180,E1 7479.692,E2 7479.692} C_VEL
LIN {X 0,Y 183.984,Z 1220.569,A -85,B 0,C 180,E1 7473.739,E2 7473.739} C_VEL
LIN {X 0,Y 184.011,Z 1220.759,A -85,B 0,C 180,E1 7468.755,E2 7468.755} C_VEL
LIN {X 0,Y 183.992,Z 1220.065,A -85,B 0,C 180,E1 7463.447,E2 7463.447} C_VEL
LIN {X 0,Y 184.352,Z 1218.349,A -85,B 0,C 180,E1 7457.788,E2 7457.788} C_VEL
LIN {X 0,Y 186.121,Z 1214.959,A -85,B 0,C 180,E1 7450.871,E2 7450.871} C_VEL
LIN {X 0,Y 189.763,Z 1209.849,A -85,B 0,C 180,E1 7444.067,E2 7444.067} C_VEL
LIN {X 0,Y 195.471,Z 1203.296,A -85,B 0,C 180,E1 7437.515,E2 7437.515} C_VEL
LIN {X 0,Y 203.247,Z 1194.879,A -85,B 0,C 180,E1 7431.335,E2 7431.335} C_VEL
LIN {X 0,Y 212.998,Z 1184.78,A -85,B 0,C 180,E1 7425.618,E2 7425.618} C_VEL
LIN {X 0,Y 223.63,Z 1173.47,A -85,B 0,C 180,E1 7420.753,E2 7420.753} C_VEL
LIN {X 0,Y 235.736,Z 1160.223,A -85,B 0,C 180,E1 7416.306,E2 7416.306} C_VEL
LIN {X 0,Y 247.328,Z 1146.734,A -85,B 0,C 180,E1 7412.768,E2 7412.768} C_VEL
LIN {X 0,Y 260.449,Z 1130.341,A -85,B 0,C 180,E1 7409.373,E2 7409.373} C_VEL
LIN {X 0,Y 272.123,Z 1114.485,A -85,B 0,C 180,E1 7406.767,E2 7406.767} C_VEL
LIN {X 0,Y 284.287,Z 1096.231,A -85,B 0,C 180,E1 7404.367,E2 7404.367} C_VEL
LIN {X 0,Y 294.862,Z 1078.693,A -85,B 0,C 180,E1 7402.503,E2 7402.503} C_VEL
LIN {X 0,Y 305.303,Z 1059.123,A -85,B 0,C 180,E1 7400.818,E2 7400.818} C_VEL
LIN {X 0,Y 314.425,Z 1039.795,A -85,B 0,C 180,E1 7399.463,E2 7399.463} C_VEL
LIN {X 0,Y 323.19,Z 1018.062,A -85,B 0,C 180,E1 7398.238,E2 7398.238} C_VEL
LIN {X 0,Y 330.807,Z 995.8,A -85,B 0,C 180,E1 7397.234,E2 7397.234} C_VEL
LIN {X 0,Y 337.078,Z 972.68,A -85,B 0,C 180,E1 7396.44,E2 7396.44} C_VEL
LIN {X 0,Y 342.1,Z 948.89,A -85,B 0,C 180,E1 7395.821,E2 7395.821} C_VEL
LIN {X 0,Y 345.377,Z 926.307,A -85,B 0,C 180,E1 7395.386,E2 7395.386} C_VEL
LIN {X 0,Y 363.063,Z 753.109,A -85,B 0,C 180,E1 7392.613,E2 7392.613} C_VEL
LIN {X 0,Y 359.349,Z 746.143,A -85,B 0,C 180,E1 7389.772,E2 7389.772} C_VEL
LIN {X 0,Y 356.526,Z 741.095,A -85,B 0,C 180,E1 7387.088,E2 7387.088} C_VEL
LIN {X 0,Y 354.059,Z 737.354,A -85,B 0,C 180,E1 7384.049,E2 7384.049} C_VEL
LIN {X 0,Y 352.151,Z 735.112,A -85,B 0,C 180,E1 7380.325,E2 7380.325} C_VEL
LIN {X 0,Y 351.437,Z 735.242,A -85,B 0,C 180,E1 7377.228,E2 7377.228} C_VEL
LIN {X 0,Y 351.612,Z 736.807,A -85,B 0,C 180,E1 7373.96,E2 7373.96} C_VEL
LIN {X 0,Y 352.622,Z 740.586,A -85,B 0,C 180,E1 7370.781,E2 7370.781} C_VEL
LIN {X 0,Y 354.087,Z 744.631,A -85,B 0,C 180,E1 7368.269,E2 7368.269} C_VEL
LIN {X 0,Y 356.634,Z 751.872,A -85,B 0,C 180,E1 7365.135,E2 7365.135} C_VEL
LIN {X 0,Y 359.046,Z 758.675,A -85,B 0,C 180,E1 7362.831,E2 7362.831} C_VEL
LIN {X 0,Y 361.22,Z 764.847,A -85,B 0,C 180,E1 7361.056,E2 7361.056} C_VEL
LIN {X 0,Y 343.957,Z 941.617,A -85,B 0,C 180,E1 7358.357,E2 7358.357} C_VEL
LIN {X 0,Y 340.026,Z 965.056,A -85,B 0,C 180,E1 7357.888,E2 7357.888} C_VEL
LIN {X 0,Y 334.826,Z 987.302,A -85,B 0,C 180,E1 7357.329,E2 7357.329} C_VEL
LIN {X 0,Y 328.426,Z 1008.276,A -85,B 0,C 180,E1 7356.618,E2 7356.618} C_VEL
LIN {X 0,Y 320.444,Z 1030.066,A -85,B 0,C 180,E1 7355.658,E2 7355.658} C_VEL
LIN {X 0,Y 312.108,Z 1049.184,A -85,B 0,C 180,E1 7354.577,E2 7354.577} C_VEL
LIN {X 0,Y 301.616,Z 1069.981,A -85,B 0,C 180,E1 7353.092,E2 7353.092} C_VEL
LIN {X 0,Y 291.317,Z 1087.897,A -85,B 0,C 180,E1 7351.479,E2 7351.479} C_VEL
LIN {X 0,Y 279.752,Z 1105.648,A -85,B 0,C 180,E1 7349.469,E2 7349.469} C_VEL
LIN {X 0,Y 267.87,Z 1122.175,A -85,B 0,C 180,E1 7347.123,E2 7347.123} C_VEL
LIN {X 0,Y 255.543,Z 1137.481,A -85,B 0,C 180,E1 7344.337,E2 7344.337} C_VEL
LIN {X 0,Y 242.666,Z 1152.207,A -85,B 0,C 180,E1 7340.918,E2 7340.918} C_VEL
LIN {X 0,Y 231.26,Z 1164.258,A -85,B 0,C 180,E1 7337.307,E2 7337.307} C_VEL
LIN {X 0,Y 219.464,Z 1175.935,A -85,B 0,C 180,E1 7332.752,E2 7332.752} C_VEL
LIN {X 0,Y 209.168,Z 1185.773,A -85,B 0,C 180,E1 7327.724,E2 7327.724} C_VEL
LIN {X 0,Y 200.159,Z 1194.039,A -85,B 0,C 180,E1 7321.972,E2 7321.972} C_VEL
LIN {X 0,Y 192.89,Z 1200.912,A -85,B 0,C 180,E1 7315.482,E2 7315.482} C_VEL
LIN {X 0,Y 188.253,Z 1205.593,A -85,B 0,C 180,E1 7309.226,E2 7309.226} C_VEL
LIN {X 0,Y 185.222,Z 1209.211,A -85,B 0,C 180,E1 7301.837,E2 7301.837} C_VEL
LIN {X 0,Y 184.218,Z 1210.9,A -85,B 0,C 180,E1 7295.607,E2 7295.607} C_VEL
LIN {X 0,Y 184.048,Z 1211.412,A -85,B 0,C 180,E1 7289.377,E2 7289.377} C_VEL
LIN {X 0,Y 184.288,Z 1210.742,A -85,B 0,C 180,E1 7283.458,E2 7283.458} C_VEL
LIN {X 0,Y 185.548,Z 1208.839,A -85,B 0,C 180,E1 7276.919,E2 7276.919} C_VEL
LIN {X 0,Y 188.75,Z 1205.105,A -85,B 0,C 180,E1 7269.86,E2 7269.86} C_VEL
LIN {X 0,Y 194.209,Z 1199.763,A -85,B 0,C 180,E1 7263.06,E2 7263.06} C_VEL
LIN {X 0,Y 201.557,Z 1192.855,A -85,B 0,C 180,E1 7256.929,E2 7256.929} C_VEL
LIN {X 0,Y 211.358,Z 1183.773,A -85,B 0,C 180,E1 7251.011,E2 7251.011} C_VEL
LIN {X 0,Y 222.026,Z 1173.679,A -85,B 0,C 180,E1 7246.091,E2 7246.091} C_VEL
LIN {X 0,Y 233.524,Z 1162.088,A -85,B 0,C 180,E1 7241.841,E2 7241.841} C_VEL
LIN {X 0,Y 245.529,Z 1149.315,A -85,B 0,C 180,E1 7238.192,E2 7238.192} C_VEL
LIN {X 0,Y 257.732,Z 1135.119,A -85,B 0,C 180,E1 7235.059,E2 7235.059} C_VEL
LIN {X 0,Y 271.01,Z 1118.194,A -85,B 0,C 180,E1 7232.145,E2 7232.145} C_VEL
LIN {X 0,Y 282.765,Z 1101.657,A -85,B 0,C 180,E1 7229.907,E2 7229.907} C_VEL
LIN {X 0,Y 294.244,Z 1083.389,A -85,B 0,C 180,E1 7227.966,E2 7227.966} C_VEL
LIN {X 0,Y 305.094,Z 1063.976,A -85,B 0,C 180,E1 7226.322,E2 7226.322} C_VEL
LIN {X 0,Y 314.487,Z 1044.582,A -85,B 0,C 180,E1 7225.027,E2 7225.027} C_VEL
LIN {X 0,Y 323.635,Z 1022.485,A -85,B 0,C 180,E1 7223.868,E2 7223.868} C_VEL
LIN {X 0,Y 330.845,Z 1001.802,A -85,B 0,C 180,E1 7223.028,E2 7223.028} C_VEL
